KUKA KRL program: MyProgram_251().src

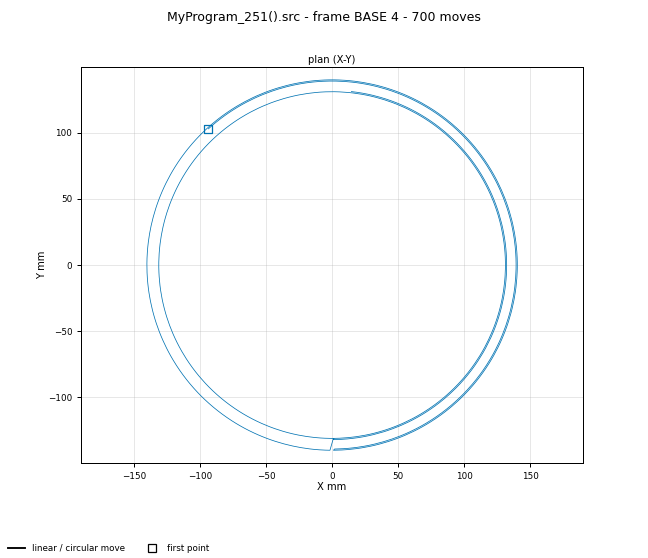
[picture p0: tool path of MyProgram_251().src in frame BASE 4, 700 of 700 moves have a stored position in this frame; points joined in program order, loops and branches not executed]
&ACCESS RVP
&REL 1
&PARAM TEMPLATE = C:\KRC\Roboter\Template\vorgabe
&PARAM EDITMASK = *
DEF MyProgram_251()
; ---- Setting reference (Base) ----
$BASE = BASE_DATA[4]

; --------------------------
; ---- Setting tool (TCP) ----
$TOOL = TOOL_DATA[3]
; --------------------------

$VEL.CP = VEL_APROX_PRINT
Startdeposition()
$VEL.CP = VEL_PRINT
LIN {X -93.5132,Y 103.0033,Z 164,A 132.083,B 11.8455,C 0.0416,E1 11.7391,E2 318.6736} C_DIS
LIN {X -90.9091,Y 105.3089,Z 164,A 130.6284,B 11.8455,C 0.0393,E1 11.7422,E2 320.1295} C_DIS
LIN {X -88.157,Y 107.6233,Z 164,A 129.1078,B 11.8455,C 0.0373,E1 11.7455,E2 321.6535} C_DIS
LIN {X -84.8361,Y 110.2606,Z 164,A 127.2395,B 11.8455,C 0.0369,E1 11.7496,E2 323.535} C_DIS
LIN {X -82.0924,Y 112.3181,Z 164,A 125.9276,B 11.8455,C 0.032,E1 11.7525,E2 324.833} C_DIS
LIN {X -78.8716,Y 114.6024,Z 164,A 124.2342,B 11.8455,C 0.0308,E1 11.7564,E2 326.5331} C_DIS
LIN {X -75.1837,Y 117.055,Z 164,A 121.9812,B 11.8455,C 0.0378,E1 11.7618,E2 328.8371} C_DIS
LIN {X -71.4051,Y 119.3975,Z 164,A 120.7033,B 11.8455,C 0.0219,E1 11.7647,E2 330.0452} C_DIS
LIN {X -67.8999,Y 121.4253,Z 164,A 118.948,B 11.8455,C 0.0214,E1 11.769,E2 331.8098} C_DIS
LIN {X -64.5496,Y 123.2364,Z 164,A 117.0261,B 11.8455,C 0.0276,E1 11.7738,E2 333.7737} C_DIS
LIN {X -61.2678,Y 124.9008,Z 164,A 115.8624,B 11.8455,C 0.0171,E1 11.7766,E2 334.8928} C_DIS
LIN {X -58.3954,Y 126.2689,Z 164,A 114.5881,B 11.8455,C 0.0145,E1 11.7798,E2 336.1615} C_DIS
LIN {X -55.0308,Y 127.7713,Z 164,A 112.9634,B 11.8455,C 0.0152,E1 11.784,E2 337.7981} C_DIS
LIN {X -51.9488,Y 129.055,Z 164,A 111.5636,B 11.8455,C 0.0142,E1 11.7877,E2 339.1998} C_DIS
LIN {X -47.7233,Y 130.6779,Z 164,A 109.8659,B 11.8456,C 0.0081,E1 11.792,E2 340.8755} C_DIS
LIN {X -45.5011,Y 131.4669,Z 164,A 108.7026,B 11.8456,C 0.0118,E1 11.7952,E2 342.0617} C_DIS
LIN {X -40.6187,Y 133.0565,Z 164,A 106.6929,B 11.8456,C 0.0072,E1 11.8005,E2 344.0567} C_DIS
LIN {X -37.3347,Y 134.0151,Z 164,A 105.2264,B 11.8456,C 0.0074,E1 11.8044,E2 345.5294} C_DIS
LIN {X -34.0868,Y 134.8778,Z 164,A 103.8149,B 11.8456,C 0.007,E1 11.8082,E2 346.9433} C_DIS
LIN {X -29.7542,Y 135.8999,Z 164,A 101.958,B 11.8456,C 0.0062,E1 11.8133,E2 348.8019} C_DIS
LIN {X -26.0587,Y 136.6561,Z 164,A 100.4689,B 11.8456,C 0.0037,E1 11.8174,E2 350.2819} C_DIS
LIN {X -22.525,Y 137.2834,Z 164,A 98.5845,B 11.8456,C 0.0129,E1 11.8227,E2 352.2155} C_DIS
LIN {X -18.6482,Y 137.8642,Z 164,A 97.4654,B 11.8456,C -0.0001,E1 11.8256,E2 353.2725} C_DIS
LIN {X -14.4572,Y 138.366,Z 164,A 95.6217,B 11.8456,C 0.0018,E1 11.8308,E2 355.1283} C_DIS
LIN {X -10.8534,Y 138.6965,Z 164,A 94.0872,B 11.8456,C 0.0025,E1 11.835,E2 356.6675} C_DIS
LIN {X -7.1224,Y 138.9363,Z 164,A 92.5483,B 11.8456,C 0.0021,E1 11.8393,E2 358.2053} C_DIS
LIN {X -1.7781,Y 139.1081,Z 164,A 90.2365,B 11.8456,C 0.0046,E1 11.8458,E2 360.5297} C_DIS
LIN {X 2.8679,Y 139.0903,Z 164,A 88.5296,B 11.8456,C -0.0007,E1 11.8505,E2 362.2101} C_DIS
LIN {X 6.3016,Y 138.9776,Z 164,A 87.1185,B 11.8456,C -0.0007,E1 11.8544,E2 363.6202} C_DIS
LIN {X 9.3557,Y 138.8057,Z 164,A 85.6308,B 11.8456,C 0.0053,E1 11.8587,E2 365.1356} C_DIS
LIN {X 15.0229,Y 138.3051,Z 164,A 83.549,B 11.8456,C -0.001,E1 11.8644,E2 367.1842} C_DIS
LIN {X 18.2395,Y 137.9178,Z 164,A 82.134,B 11.8456,C 0.0015,E1 11.8683,E2 368.6087} C_DIS
LIN {X 21.7401,Y 137.4101,Z 164,A 80.0938,B 11.8456,C 0.0172,E1 11.8741,E2 370.7205} C_DIS
LIN {X 26.5047,Y 136.5709,Z 164,A 78.6953,B 11.8456,C 0.0028,E1 11.8778,E2 372.0452} C_DIS
LIN {X 30.1426,Y 135.8161,Z 164,A 77.0002,B 11.8456,C 0.0079,E1 11.8825,E2 373.7605} C_DIS
LIN {X 34.389,Y 134.8012,Z 164,A 75.2809,B 11.8456,C 0.007,E1 11.8871,E2 375.4696} C_DIS
LIN {X 38.2782,Y 133.7512,Z 164,A 73.7125,B 11.8456,C 0.0059,E1 11.8913,E2 377.0265} C_DIS
LIN {X 41.1605,Y 132.8907,Z 164,A 72.462,B 11.8456,C 0.0072,E1 11.8946,E2 378.2782} C_DIS
LIN {X 45.0474,Y 131.6242,Z 164,A 70.7128,B 11.8456,C 0.0104,E1 11.8993,E2 380.0355} C_DIS
LIN {X 48.204,Y 130.5016,Z 164,A 69.5013,B 11.8456,C 0.0072,E1 11.9024,E2 381.2259} C_DIS
LIN {X 50.6781,Y 129.5596,Z 164,A 68.3915,B 11.8456,C 0.0088,E1 11.9053,E2 382.338} C_DIS
LIN {X 53.1807,Y 128.5531,Z 164,A 67.3491,B 11.8456,C 0.0082,E1 11.908,E2 383.3718} C_DIS
LIN {X 57.2624,Y 126.7878,Z 164,A 65.4033,B 11.8456,C 0.0133,E1 11.913,E2 385.3319} C_DIS
LIN {X 60.3441,Y 125.35,Z 164,A 63.9218,B 11.8456,C 0.0172,E1 11.9168,E2 386.8236} C_DIS
LIN {X 64.3775,Y 123.3268,Z 164,A 62.1382,B 11.8456,C 0.0175,E1 11.9212,E2 388.598} C_DIS
LIN {X 68.1253,Y 121.2986,Z 164,A 60.3486,B 11.8456,C 0.0209,E1 11.9256,E2 390.3922} C_DIS
LIN {X 71.8558,Y 119.1267,Z 164,A 58.6255,B 11.8456,C 0.022,E1 11.9297,E2 392.1087} C_DIS
LIN {X 75.3059,Y 116.9767,Z 164,A 56.8769,B 11.8456,C 0.0266,E1 11.9338,E2 393.8669} C_DIS
LIN {X 79.1791,Y 114.3905,Z 164,A 55.0231,B 11.8456,C 0.0279,E1 11.9381,E2 395.7131} C_DIS
LIN {X 82.2792,Y 112.1809,Z 164,A 53.4542,B 11.8456,C 0.0305,E1 11.9416,E2 397.2825} C_DIS
LIN {X 85.5645,Y 109.6965,Z 164,A 51.786,B 11.8456,C 0.0327,E1 11.9453,E2 398.9477} C_DIS
LIN {X 88.6989,Y 107.177,Z 164,A 50.0509,B 11.8456,C 0.0379,E1 11.9491,E2 400.6931} C_DIS
LIN {X 91.429,Y 104.8578,Z 164,A 48.639,B 11.8456,C 0.0389,E1 11.9521,E2 402.0976} C_DIS
LIN {X 94.8874,Y 101.7389,Z 164,A 46.6702,B 11.8456,C 0.0441,E1 11.9561,E2 404.0735} C_DIS
LIN {X 97.912,Y 98.8317,Z 164,A 45.0073,B 11.8456,C 0.0457,E1 11.9595,E2 405.729} C_DIS
LIN {X 101.1689,Y 95.4948,Z 164,A 42.6719,B 11.8454,C 0.0613,E1 11.9641,E2 408.1169} C_DIS
LIN {X 104.3624,Y 91.9942,Z 164,A 41.1925,B 11.8454,C 0.0524,E1 11.9667,E2 409.5385} C_DIS
LIN {X 107.3104,Y 88.5379,Z 164,A 39.3371,B 11.8454,C 0.0561,E1 11.97,E2 411.3929} C_DIS
LIN {X 109.9995,Y 85.1735,Z 164,A 37.6211,B 11.8454,C 0.0585,E1 11.973,E2 413.1027} C_DIS
LIN {X 112.4762,Y 81.8755,Z 164,A 35.9215,B 11.8454,C 0.0625,E1 11.9758,E2 414.8033} C_DIS
LIN {X 114.8679,Y 78.4848,Z 164,A 34.1903,B 11.8454,C 0.0672,E1 11.9786,E2 416.5384} C_DIS
LIN {X 117.2497,Y 74.8796,Z 164,A 32.3977,B 11.8454,C 0.0719,E1 11.9813,E2 418.3338} C_DIS
LIN {X 120.2343,Y 69.9875,Z 164,A 29.8739,B 11.8454,C 0.0824,E1 11.9849,E2 420.8797} C_DIS
LIN {X 121.9796,Y 66.8991,Z 164,A 28.9447,B 11.8454,C 0.071,E1 11.9861,E2 421.7431} C_DIS
LIN {X 123.3941,Y 64.2493,Z 164,A 27.5566,B 11.8454,C 0.0785,E1 11.9879,E2 423.1511} C_DIS
LIN {X 124.8289,Y 61.4135,Z 164,A 26.2825,B 11.8454,C 0.0809,E1 11.9895,E2 424.4218} C_DIS
LIN {X 126.5429,Y 57.8029,Z 164,A 24.4503,B 11.8453,C 0.0906,E1 11.9917,E2 426.2788} C_DIS
LIN {X 129.4436,Y 50.9761,Z 164,A 21.3576,B 11.8452,C 0.0999,E1 11.995,E2 429.3787} C_DIS
LIN {X 131.0516,Y 46.6866,Z 164,A 19.7563,B 11.8452,C 0.0969,E1 11.9965,E2 430.9456} C_DIS
LIN {X 131.9741,Y 44.0084,Z 164,A 18.5216,B 11.8452,C 0.1021,E1 11.9976,E2 432.1899} C_DIS
LIN {X 133.2683,Y 39.9269,Z 164,A 16.8422,B 11.8452,C 0.1046,E1 11.999,E2 433.8604} C_DIS
LIN {X 134.1255,Y 36.94,Z 164,A 15.5694,B 11.8452,C 0.108,E1 12,E2 435.1334} C_DIS
LIN {X 134.9661,Y 33.7389,Z 164,A 14.2687,B 11.8451,C 0.1101,E1 12.0009,E2 436.4275} C_DIS
LIN {X 135.6818,Y 30.7319,Z 164,A 12.9918,B 11.8451,C 0.1138,E1 12.0017,E2 437.706} C_DIS
LIN {X 136.5733,Y 26.4921,Z 164,A 11.3784,B 11.8451,C 0.114,E1 12.0026,E2 439.2995} C_DIS
LIN {X 137.6895,Y 19.8898,Z 164,A 8.3669,B 11.8449,C 0.1294,E1 12.004,E2 442.3459} C_DIS
LIN {X 138.4064,Y 14.0802,Z 164,A 6.13,B 11.8449,C 0.1314,E1 12.0047,E2 444.5633} C_DIS
LIN {X 138.8292,Y 8.9791,Z 164,A 3.8602,B 11.8448,C 0.1423,E1 12.0052,E2 446.8558} C_DIS
LIN {X 139.0245,Y 5.1275,Z 164,A 2.3451,B 11.8448,C 0.1448,E1 12.0053,E2 448.3632} C_DIS
LIN {X 139.1177,Y 0.5934,Z 164,A 0.6055,B 11.8448,C 0.1466,E1 12.0054,E2 450.0885} C_DIS
LIN {X 139.0869,Y -3.0686,Z 164,A -1.0543,B 11.8446,C 0.1555,E1 12.0054,E2 451.7693} C_DIS
LIN {X 138.9554,Y -6.7431,Z 164,A -2.2689,B 11.8446,C 0.1512,E1 12.0052,E2 452.9474} C_DIS
LIN {X 138.8089,Y -9.3088,Z 164,A -3.4315,B 11.8446,C 0.1574,E1 12.005,E2 454.1245} C_DIS
LIN {X 138.443,Y -13.7002,Z 164,A -5.0964,B 11.8446,C 0.1584,E1 12.0046,E2 455.7722} C_DIS
LIN {X 138.1355,Y -16.5095,Z 164,A -6.3924,B 11.8445,C 0.1657,E1 12.0042,E2 457.0864} C_DIS
LIN {X 137.6077,Y -20.4623,Z 164,A -8.0526,B 11.8444,C 0.171,E1 12.0035,E2 458.7507} C_DIS
LIN {X 137.0427,Y -23.9491,Z 164,A -9.9366,B 11.8441,C 0.1878,E1 12.0026,E2 460.6908} C_DIS
LIN {X 136.1753,Y -28.4745,Z 164,A -11.2702,B 11.8443,C 0.1769,E1 12.0019,E2 461.9551} C_DIS
LIN {X 135.5749,Y -31.1998,Z 164,A -12.4598,B 11.8443,C 0.1814,E1 12.0012,E2 463.1511} C_DIS
LIN {X 134.6428,Y -35.0126,Z 164,A -14.1607,B 11.8441,C 0.1886,E1 12,E2 464.8647} C_DIS
LIN {X 133.4452,Y -39.3237,Z 164,A -15.8891,B 11.8441,C 0.1905,E1 11.9987,E2 466.5806} C_DIS
LIN {X 132.2596,Y -43.1508,Z 164,A -17.4741,B 11.8441,C 0.1933,E1 11.9973,E2 468.1593} C_DIS
LIN {X 131.3169,Y -45.9338,Z 164,A -18.779,B 11.8439,C 0.1995,E1 11.9961,E2 469.4777} C_DIS
LIN {X 129.7349,Y -50.2272,Z 164,A -20.3354,B 11.844,C 0.1952,E1 11.9947,E2 470.9943} C_DIS
LIN {X 128.9064,Y -52.3176,Z 164,A -21.5007,B 11.8439,C 0.2048,E1 11.9934,E2 472.1913} C_DIS
LIN {X 127.3612,Y -55.9795,Z 164,A -23.075,B 11.8439,C 0.2075,E1 11.9917,E2 473.7596} C_DIS
LIN {X 125.8906,Y -59.2126,Z 164,A -24.5095,B 11.8438,C 0.2107,E1 11.99,E2 475.1922} C_DIS
LIN {X 123.5041,Y -64.0398,Z 164,A -26.6881,B 11.8437,C 0.2155,E1 11.9873,E2 477.3685} C_DIS
LIN {X 121.613,Y -67.5628,Z 164,A -28.4394,B 11.8435,C 0.2229,E1 11.9849,E2 479.1351} C_DIS
LIN {X 119.3266,Y -71.5241,Z 164,A -30.4512,B 11.8434,C 0.2315,E1 11.982,E2 481.1655} C_DIS
LIN {X 116.6984,Y -75.7357,Z 164,A -32.7824,B 11.8431,C 0.245,E1 11.9785,E2 483.5355} C_DIS
LIN {X 113.9889,Y -79.7564,Z 164,A -34.5272,B 11.8431,C 0.2427,E1 11.9757,E2 485.2506} C_DIS
LIN {X 111.9253,Y -82.6271,Z 164,A -35.7711,B 11.8432,C 0.2402,E1 11.9737,E2 486.4691} C_DIS
LIN {X 108.9221,Y -86.5471,Z 164,A -37.6893,B 11.8432,C 0.2418,E1 11.9704,E2 488.3748} C_DIS
LIN {X 106.4676,Y -89.5493,Z 164,A -39.2737,B 11.8432,C 0.2452,E1 11.9676,E2 489.9594} C_DIS
LIN {X 103.9721,Y -92.4357,Z 164,A -40.8028,B 11.8431,C 0.2476,E1 11.9648,E2 491.4849} C_DIS
LIN {X 102.2519,Y -94.3346,Z 164,A -41.8981,B 11.843,C 0.2511,E1 11.9627,E2 492.5865} C_DIS
LIN {X 99.3369,Y -97.3991,Z 164,A -43.6258,B 11.843,C 0.2546,E1 11.9594,E2 494.3143} C_DIS
LIN {X 96.2847,Y -100.4177,Z 164,A -45.38,B 11.8428,C 0.258,E1 11.9559,E2 496.0687} C_DIS
LIN {X 93.0721,Y -103.4026,Z 164,A -47.1893,B 11.8428,C 0.2619,E1 11.9521,E2 497.8804} C_DIS
LIN {X 89.8236,Y -106.2368,Z 164,A -48.9498,B 11.8427,C 0.265,E1 11.9484,E2 499.6408} C_DIS
LIN {X 86.4839,Y -108.9724,Z 164,A -50.7,B 11.8427,C 0.2677,E1 11.9446,E2 501.3894} C_DIS
LIN {X 82.9756,Y -111.6668,Z 164,A -52.5243,B 11.8425,C 0.2712,E1 11.9405,E2 503.2158} C_DIS
LIN {X 79.1848,Y -114.3866,Z 164,A -54.4412,B 11.8425,C 0.2746,E1 11.9362,E2 505.1341} C_DIS
LIN {X 75.5705,Y -116.8057,Z 164,A -56.1855,B 11.8425,C 0.2764,E1 11.9321,E2 506.8742} C_DIS
LIN {X 71.1252,Y -119.5643,Z 164,A -58.2357,B 11.8425,C 0.277,E1 11.9272,E2 508.913} C_DIS
LIN {X 67.8853,Y -121.4335,Z 164,A -59.88,B 11.8423,C 0.2823,E1 11.9232,E2 510.5722} C_DIS
LIN {X 63.8811,Y -123.5872,Z 164,A -61.6454,B 11.8423,C 0.2821,E1 11.9189,E2 512.3255} C_DIS
LIN {X 58.7901,Y -126.0864,Z 164,A -63.8155,B 11.8423,C 0.2808,E1 11.9135,E2 514.4764} C_DIS
LIN {X 55.0946,Y -127.7438,Z 164,A -65.6415,B 11.8422,C 0.2874,E1 11.9088,E2 516.3242} C_DIS
LIN {X 51.7597,Y -129.1313,Z 164,A -67.194,B 11.8421,C 0.291,E1 11.9047,E2 517.8863} C_DIS
LIN {X 48.2107,Y -130.4991,Z 164,A -68.6428,B 11.8421,C 0.2896,E1 11.901,E2 519.3213} C_DIS
LIN {X 45.2496,Y -131.5541,Z 164,A -70.0506,B 11.8421,C 0.2942,E1 11.8972,E2 520.7447} C_DIS
LIN {X 41.6349,Y -132.744,Z 164,A -71.4992,B 11.8421,C 0.2926,E1 11.8934,E2 522.1794} C_DIS
LIN {X 38.929,Y -133.5607,Z 164,A -72.6474,B 11.8421,C 0.2932,E1 11.8903,E2 523.3264} C_DIS
LIN {X 35.3733,Y -134.547,Z 164,A -74.1782,B 11.842,C 0.2949,E1 11.8862,E2 524.8597} C_DIS
LIN {X 32.2595,Y -135.3269,Z 164,A -75.4773,B 11.842,C 0.2954,E1 11.8827,E2 526.1569} C_DIS
LIN {X 28.5095,Y -136.1682,Z 164,A -77.5593,B 11.8416,C 0.31,E1 11.8768,E2 528.3038} C_DIS
LIN {X 24.3803,Y -136.9656,Z 164,A -78.9498,B 11.8418,C 0.302,E1 11.8731,E2 529.6518} C_DIS
LIN {X 18.9709,Y -137.8208,Z 164,A -81.0414,B 11.8418,C 0.2989,E1 11.8674,E2 531.7239} C_DIS
LIN {X 15.8743,Y -138.2113,Z 164,A -82.7304,B 11.8416,C 0.3103,E1 11.8626,E2 533.4653} C_DIS
LIN {X 12.0921,Y -138.5926,Z 164,A -84.0223,B 11.8418,C 0.3037,E1 11.8591,E2 534.7231} C_DIS
LIN {X 8.5469,Y -138.8559,Z 164,A -85.456,B 11.8418,C 0.3033,E1 11.8551,E2 536.1537} C_DIS
LIN {X 4.8994,Y -139.0334,Z 164,A -86.8146,B 11.8418,C 0.2999,E1 11.8513,E2 537.4945} C_DIS
LIN {X 1.8653,Y -139.107,Z 164,A -88.1849,B 11.8418,C 0.3033,E1 11.8475,E2 538.8809} C_DIS
LIN {X 1.8653,Y -139.107,Z 164,A -88.1849,B 11.8418,C 0.3033,E1 11.8475,E2 538.8809} C_DIS
Enddeposition()
LIN {X 1.0011,Y -140.0329,Z 164,A -87.9487,B 11.842,C 0.2948,E1 11.8483,E2 538.6034} C_DIS
Startdeposition()
$VEL.CP = VEL_PRINT
LIN {X 4.0661,Y -139.9794,Z 164,A -86.5813,B 11.8421,C 0.2915,E1 11.8522,E2 537.2207} C_DIS
LIN {X 7.3718,Y -139.8446,Z 164,A -85.0824,B 11.8422,C 0.2872,E1 11.8564,E2 535.702} C_DIS
LIN {X 12.0541,Y -139.5188,Z 164,A -83.2838,B 11.8422,C 0.2898,E1 11.8614,E2 533.9183} C_DIS
LIN {X 15.6406,Y -139.1636,Z 164,A -81.8412,B 11.8422,C 0.29,E1 11.8654,E2 532.4791} C_DIS
LIN {X 18.9541,Y -138.7517,Z 164,A -80.3719,B 11.8422,C 0.2865,E1 11.8695,E2 530.9954} C_DIS
LIN {X 22.2682,Y -138.2586,Z 164,A -79.0797,B 11.8422,C 0.2879,E1 11.873,E2 529.7126} C_DIS
LIN {X 25.6653,Y -137.6676,Z 164,A -77.6805,B 11.8422,C 0.2873,E1 11.8768,E2 528.314} C_DIS
LIN {X 29.0223,Y -136.9988,Z 164,A -76.2843,B 11.8422,C 0.2863,E1 11.8807,E2 526.9174} C_DIS
LIN {X 32.3823,Y -136.2433,Z 164,A -74.8831,B 11.8422,C 0.2854,E1 11.8845,E2 525.5162} C_DIS
LIN {X 35.7212,Y -135.406,Z 164,A -73.4347,B 11.8423,C 0.2831,E1 11.8884,E2 524.0615} C_DIS
LIN {X 39.0397,Y -134.4866,Z 164,A -72.0852,B 11.8423,C 0.2834,E1 11.892,E2 522.7187} C_DIS
LIN {X 42.3077,Y -133.4945,Z 164,A -70.6887,B 11.8423,C 0.282,E1 11.8957,E2 521.3212} C_DIS
LIN {X 45.5732,Y -132.4152,Z 164,A -69.2884,B 11.8423,C 0.2807,E1 11.8995,E2 519.9207} C_DIS
LIN {X 48.8112,Y -131.2562,Z 164,A -67.8889,B 11.8424,C 0.2793,E1 11.9031,E2 518.5211} C_DIS
LIN {X 52.0199,Y -130.0179,Z 164,A -66.4897,B 11.8424,C 0.2779,E1 11.9068,E2 517.1217} C_DIS
LIN {X 55.1975,Y -128.7012,Z 164,A -65.0964,B 11.8424,C 0.2765,E1 11.9103,E2 515.729} C_DIS
LIN {X 58.3787,Y -127.2899,Z 164,A -63.6912,B 11.8425,C 0.2751,E1 11.9139,E2 514.3251} C_DIS
LIN {X 61.4407,Y -125.841,Z 164,A -62.301,B 11.8425,C 0.273,E1 11.9174,E2 512.933} C_DIS
LIN {X 64.5115,Y -124.2952,Z 164,A -60.9185,B 11.8425,C 0.2717,E1 11.9209,E2 511.5524} C_DIS
LIN {X 67.544,Y -122.6746,Z 164,A -59.4693,B 11.8427,C 0.2683,E1 11.9244,E2 510.0963} C_DIS
LIN {X 71.2578,Y -120.5554,Z 164,A -57.7572,B 11.8427,C 0.2666,E1 11.9286,E2 508.3875} C_DIS
LIN {X 74.4296,Y -118.6234,Z 164,A -56.1383,B 11.8428,C 0.2612,E1 11.9324,E2 506.7541} C_DIS
LIN {X 78.2094,Y -116.166,Z 164,A -54.3438,B 11.8428,C 0.2594,E1 11.9366,E2 504.9642} C_DIS
LIN {X 81.8544,Y -113.6273,Z 164,A -52.5667,B 11.8429,C 0.2573,E1 11.9406,E2 503.1906} C_DIS
LIN {X 84.813,Y -111.4361,Z 164,A -51.1314,B 11.8429,C 0.2565,E1 11.9438,E2 501.7631} C_DIS
LIN {X 87.5061,Y -109.3341,Z 164,A -49.6095,B 11.8431,C 0.2502,E1 11.9472,E2 500.2235} C_DIS
LIN {X 91.0025,Y -106.4417,Z 164,A -47.7743,B 11.8431,C 0.2471,E1 11.9511,E2 498.3891} C_DIS
LIN {X 94.4857,Y -103.3621,Z 164,A -45.953,B 11.8431,C 0.2455,E1 11.9549,E2 496.5763} C_DIS
LIN {X 97.1954,Y -100.818,Z 164,A -44.378,B 11.8432,C 0.2407,E1 11.9581,E2 494.9925} C_DIS
LIN {X 100.2454,Y -97.7862,Z 164,A -42.7214,B 11.8432,C 0.2399,E1 11.9613,E2 493.3475} C_DIS
LIN {X 103.184,Y -94.6795,Z 164,A -40.9463,B 11.8434,C 0.2352,E1 11.9647,E2 491.5671} C_DIS
LIN {X 106.0445,Y -91.4643,Z 164,A -39.1946,B 11.8434,C 0.2314,E1 11.9679,E2 489.8145} C_DIS
LIN {X 108.8027,Y -88.1658,Z 164,A -37.5509,B 11.8434,C 0.2306,E1 11.9708,E2 488.184} C_DIS
LIN {X 111.2882,Y -85.0063,Z 164,A -35.8382,B 11.8436,C 0.2247,E1 11.9738,E2 486.4605} C_DIS
LIN {X 114.0144,Y -81.3135,Z 164,A -33.9826,B 11.8436,C 0.2207,E1 11.9768,E2 484.6057} C_DIS
LIN {X 116.4423,Y -77.7967,Z 164,A -32.2283,B 11.8437,C 0.2161,E1 11.9796,E2 482.8485} C_DIS
LIN {X 118.7733,Y -74.1897,Z 164,A -30.5934,B 11.8437,C 0.2152,E1 11.982,E2 481.2276} C_DIS
LIN {X 120.5616,Y -71.2473,Z 164,A -29.2021,B 11.8437,C 0.2121,E1 11.984,E2 479.837} C_DIS
LIN {X 122.2757,Y -68.2639,Z 164,A -27.8008,B 11.8438,C 0.2086,E1 11.9859,E2 478.4348} C_DIS
LIN {X 124.0773,Y -64.9264,Z 164,A -26.3319,B 11.8438,C 0.2069,E1 11.9878,E2 476.9749} C_DIS
LIN {X 125.483,Y -62.1664,Z 164,A -25.0269,B 11.844,C 0.2023,E1 11.9895,E2 475.6634} C_DIS
LIN {X 126.9611,Y -59.0896,Z 164,A -23.6411,B 11.844,C 0.1989,E1 11.9911,E2 474.2774} C_DIS
LIN {X 128.3961,Y -55.9032,Z 164,A -22.2202,B 11.844,C 0.1952,E1 11.9927,E2 472.856} C_DIS
LIN {X 129.7483,Y -52.6888,Z 164,A -20.8116,B 11.8441,C 0.1918,E1 11.9942,E2 471.448} C_DIS
LIN {X 131.0142,Y -49.4571,Z 164,A -19.4104,B 11.8441,C 0.1884,E1 11.9956,E2 470.0476} C_DIS
LIN {X 132.1942,Y -46.2107,Z 164,A -18.0021,B 11.8442,C 0.1845,E1 11.997,E2 468.6384} C_DIS
LIN {X 133.29,Y -42.9479,Z 164,A -16.6248,B 11.8442,C 0.1814,E1 11.9982,E2 467.2634} C_DIS
LIN {X 134.3017,Y -39.671,Z 164,A -15.2396,B 11.8443,C 0.1779,E1 11.9993,E2 465.8789} C_DIS
LIN {X 135.2298,Y -36.3818,Z 164,A -13.8591,B 11.8443,C 0.1744,E1 12.0003,E2 464.499} C_DIS
LIN {X 136.0738,Y -33.0855,Z 164,A -12.4855,B 11.8444,C 0.171,E1 12.0012,E2 463.1263} C_DIS
LIN {X 136.8606,Y -29.6623,Z 164,A -11.0984,B 11.8444,C 0.1683,E1 12.0021,E2 461.744} C_DIS
LIN {X 137.5057,Y -26.5124,Z 164,A -9.7798,B 11.8445,C 0.1643,E1 12.0028,E2 460.4235} C_DIS
LIN {X 138.0567,Y -23.4777,Z 164,A -8.6616,B 11.8445,C 0.1649,E1 12.0033,E2 459.3225} C_DIS
LIN {X 138.5281,Y -20.5222,Z 164,A -7.2952,B 11.8446,C 0.1571,E1 12.0039,E2 457.9363} C_DIS
LIN {X 139.0402,Y -16.6892,Z 164,A -5.7109,B 11.8446,C 0.1524,E1 12.0045,E2 456.3499} C_DIS
LIN {X 139.4224,Y -13.1212,Z 164,A -4.3109,B 11.8447,C 0.1501,E1 12.0049,E2 454.9572} C_DIS
LIN {X 139.6938,Y -9.8232,Z 164,A -2.8259,B 11.8448,C 0.1422,E1 12.0052,E2 453.4536} C_DIS
LIN {X 139.9446,Y -5.1342,Z 164,A -1.0609,B 11.8448,C 0.1411,E1 12.0054,E2 451.7067} C_DIS
LIN {X 140.0311,Y -1.6039,Z 164,A 0.4767,B 11.8449,C 0.1341,E1 12.0054,E2 450.1556} C_DIS
LIN {X 140.0178,Y 2.3995,Z 164,A 1.9711,B 11.8449,C 0.1335,E1 12.0054,E2 448.678} C_DIS
LIN {X 139.9217,Y 5.7199,Z 164,A 3.3076,B 11.8449,C 0.1302,E1 12.0053,E2 447.343} C_DIS
LIN {X 139.6938,Y 9.8232,Z 164,A 4.9783,B 11.845,C 0.1256,E1 12.005,E2 445.672} C_DIS
LIN {X 139.3653,Y 13.7165,Z 164,A 6.5723,B 11.845,C 0.121,E1 12.0046,E2 444.0769} C_DIS
LIN {X 138.9675,Y 17.2987,Z 164,A 8.0038,B 11.845,C 0.118,E1 12.0041,E2 442.6496} C_DIS
LIN {X 138.4725,Y 20.8891,Z 164,A 9.3879,B 11.845,C 0.1166,E1 12.0036,E2 441.2766} C_DIS
LIN {X 137.9729,Y 23.9718,Z 164,A 10.7556,B 11.8452,C 0.1102,E1 12.0029,E2 439.8961} C_DIS
LIN {X 137.3429,Y 27.3482,Z 164,A 12.1426,B 11.8452,C 0.1067,E1 12.0022,E2 438.5101} C_DIS
LIN {X 136.6336,Y 30.6945,Z 164,A 13.5971,B 11.8452,C 0.101,E1 12.0013,E2 437.0471} C_DIS
LIN {X 135.8381,Y 34.0415,Z 164,A 14.9103,B 11.8452,C 0.0998,E1 12.0005,E2 435.7448} C_DIS
LIN {X 134.8789,Y 37.6608,Z 164,A 16.3541,B 11.8452,C 0.0981,E1 11.9994,E2 434.311} C_DIS
LIN {X 134.0008,Y 40.6759,Z 164,A 17.6916,B 11.8453,C 0.0929,E1 11.9983,E2 432.9656} C_DIS
LIN {X 132.9613,Y 43.9545,Z 164,A 19.0814,B 11.8453,C 0.0895,E1 11.9972,E2 431.5767} C_DIS
LIN {X 131.8417,Y 47.2066,Z 164,A 20.4792,B 11.8453,C 0.0859,E1 11.9959,E2 430.1789} C_DIS
LIN {X 130.6397,Y 50.4379,Z 164,A 21.8643,B 11.8453,C 0.0828,E1 11.9945,E2 428.796} C_DIS
LIN {X 129.3643,Y 53.6248,Z 164,A 23.2505,B 11.8453,C 0.0795,E1 11.993,E2 427.4109} C_DIS
LIN {X 128.0141,Y 56.7731,Z 164,A 24.6345,B 11.8454,C 0.0763,E1 11.9915,E2 426.0281} C_DIS
LIN {X 126.5828,Y 59.8969,Z 164,A 26.0177,B 11.8454,C 0.0732,E1 11.9899,E2 424.6467} C_DIS
LIN {X 125.0848,Y 62.9664,Z 164,A 27.4051,B 11.8454,C 0.0699,E1 11.9881,E2 423.2595} C_DIS
LIN {X 123.5011,Y 66.0205,Z 164,A 28.8037,B 11.8454,C 0.0665,E1 11.9863,E2 421.8611} C_DIS
LIN {X 121.8363,Y 69.0451,Z 164,A 30.1977,B 11.8454,C 0.0635,E1 11.9844,E2 420.4685} C_DIS
LIN {X 120.1015,Y 72.0202,Z 164,A 31.6257,B 11.8455,C 0.0594,E1 11.9824,E2 419.0371} C_DIS
LIN {X 117.8374,Y 75.6672,Z 164,A 33.4042,B 11.8455,C 0.0544,E1 11.9797,E2 417.2546} C_DIS
LIN {X 115.4743,Y 79.2264,Z 164,A 35.1614,B 11.8455,C 0.05,E1 11.977,E2 415.495} C_DIS
LIN {X 112.9875,Y 82.7346,Z 164,A 36.8825,B 11.8455,C 0.0469,E1 11.9742,E2 413.7778} C_DIS
LIN {X 110.3941,Y 86.1653,Z 164,A 38.5503,B 11.8455,C 0.0455,E1 11.9713,E2 412.1209} C_DIS
LIN {X 108.1182,Y 89.0043,Z 164,A 40.1507,B 11.8455,C 0.039,E1 11.9685,E2 410.5053} C_DIS
LIN {X 105.1528,Y 92.4886,Z 164,A 41.957,B 11.8456,C 0.0368,E1 11.9652,E2 408.7065} C_DIS
LIN {X 102.1494,Y 95.7956,Z 164,A 43.7304,B 11.8456,C 0.0344,E1 11.9619,E2 406.9392} C_DIS
LIN {X 99.6254,Y 98.4179,Z 164,A 45.1621,B 11.8456,C 0.033,E1 11.9591,E2 405.5141} C_DIS
LIN {X 97.1779,Y 100.8349,Z 164,A 46.6112,B 11.8456,C 0.029,E1 11.9562,E2 404.0591} C_DIS
LIN {X 94.0343,Y 103.7723,Z 164,A 48.3899,B 11.8456,C 0.025,E1 11.9525,E2 402.2775} C_DIS
LIN {X 90.8018,Y 106.6123,Z 164,A 50.1534,B 11.8456,C 0.0216,E1 11.9488,E2 400.5129} C_DIS
LIN {X 87.5052,Y 109.3349,Z 164,A 51.781,B 11.8456,C 0.0219,E1 11.9453,E2 398.9004} C_DIS
LIN {X 84.2284,Y 111.8782,Z 164,A 53.5432,B 11.8456,C 0.0171,E1 11.9414,E2 397.1293} C_DIS
LIN {X 80.6289,Y 114.4994,Z 164,A 55.3622,B 11.8456,C 0.0142,E1 11.9372,E2 395.3103} C_DIS
LIN {X 77.074,Y 116.922,Z 164,A 57.1302,B 11.8456,C 0.0111,E1 11.9331,E2 393.5409} C_DIS
LIN {X 73.4459,Y 119.2347,Z 164,A 58.7726,B 11.8456,C 0.0118,E1 11.9293,E2 391.9132} C_DIS
LIN {X 70.4949,Y 121.0031,Z 164,A 60.1681,B 11.8456,C 0.0101,E1 11.9259,E2 390.5191} C_DIS
LIN {X 67.5221,Y 122.6867,Z 164,A 61.5688,B 11.8456,C 0.008,E1 11.9225,E2 389.1178} C_DIS
LIN {X 64.4876,Y 124.3077,Z 164,A 62.9964,B 11.8456,C 0.0056,E1 11.919,E2 387.6875} C_DIS
LIN {X 61.1115,Y 126.0026,Z 164,A 64.6366,B 11.8456,C 0.0011,E1 11.9148,E2 386.0352} C_DIS
LIN {X 57.5135,Y 127.6829,Z 164,A 66.1261,B 11.8456,C 0.0029,E1 11.9111,E2 384.5628} C_DIS
LIN {X 54.2997,Y 129.0824,Z 164,A 67.5486,B 11.8456,C 0.0016,E1 11.9074,E2 383.1418} C_DIS
LIN {X 51.0779,Y 130.3909,Z 164,A 68.9641,B 11.8456,C 0.0004,E1 11.9038,E2 381.7273} C_DIS
LIN {X 47.8376,Y 131.6142,Z 164,A 70.3745,B 11.8456,C -0.0008,E1 11.9001,E2 380.3178} C_DIS
LIN {X 44.5798,Y 132.7531,Z 164,A 71.7801,B 11.8456,C -0.0019,E1 11.8964,E2 378.9131} C_DIS
LIN {X 41.3072,Y 133.8075,Z 164,A 73.2378,B 11.8456,C -0.0045,E1 11.8925,E2 377.4491} C_DIS
LIN {X 37.3328,Y 134.9706,Z 164,A 74.8872,B 11.8456,C -0.0045,E1 11.8881,E2 375.8057} C_DIS
LIN {X 33.7943,Y 135.9009,Z 164,A 76.3563,B 11.8456,C -0.0048,E1 11.8841,E2 374.3404} C_DIS
LIN {X 30.4913,Y 136.6801,Z 164,A 77.8112,B 11.8456,C -0.0074,E1 11.8801,E2 372.8774} C_DIS
LIN {X 26.5137,Y 137.5054,Z 164,A 79.3913,B 11.8456,C -0.0061,E1 11.8758,E2 371.3081} C_DIS
LIN {X 23.4452,Y 138.0622,Z 164,A 80.5265,B 11.8456,C -0.0029,E1 11.8727,E2 370.191} C_DIS
LIN {X 20.5335,Y 138.5265,Z 164,A 81.8972,B 11.8456,C -0.0077,E1 11.8689,E2 368.7999} C_DIS
LIN {X 17.1045,Y 138.9907,Z 164,A 83.3673,B 11.8456,C -0.0096,E1 11.8648,E2 367.3234} C_DIS
LIN {X 13.1184,Y 139.4227,Z 164,A 84.9212,B 11.8456,C -0.0078,E1 11.8605,E2 365.781} C_DIS
LIN {X 9.8203,Y 139.694,Z 164,A 86.4239,B 11.8456,C -0.0119,E1 11.8563,E2 364.2601} C_DIS
LIN {X 5.1216,Y 139.945,Z 164,A 88.2135,B 11.8456,C -0.0085,E1 11.8513,E2 362.4884} C_DIS
LIN {X 1.6056,Y 140.031,Z 164,A 89.7805,B 11.8456,C -0.0118,E1 11.8469,E2 360.9059} C_DIS
LIN {X -2.3939,Y 140.0179,Z 164,A 91.2798,B 11.8456,C -0.0081,E1 11.8428,E2 359.4246} C_DIS
LIN {X -5.7206,Y 139.9217,Z 164,A 92.6362,B 11.8456,C -0.0077,E1 11.839,E2 358.0696} C_DIS
LIN {X -9.8203,Y 139.694,Z 164,A 94.4421,B 11.8456,C -0.0106,E1 11.8339,E2 356.2487} C_DIS
LIN {X -13.9852,Y 139.3395,Z 164,A 96.0303,B 11.8456,C -0.0069,E1 11.8296,E2 354.6768} C_DIS
LIN {X -17.3002,Y 138.9673,Z 164,A 97.5131,B 11.8456,C -0.0093,E1 11.8254,E2 353.18} C_DIS
LIN {X -20.9656,Y 138.4606,Z 164,A 98.7994,B 11.8456,C -0.0028,E1 11.8219,E2 351.9233} C_DIS
LIN {X -23.9569,Y 137.9756,Z 164,A 100.1858,B 11.8456,C -0.0058,E1 11.8181,E2 350.5193} C_DIS
LIN {X -27.3416,Y 137.3443,Z 164,A 101.5945,B 11.8456,C -0.005,E1 11.8142,E2 349.1115} C_DIS
LIN {X -30.7073,Y 136.6307,Z 164,A 103.0041,B 11.8456,C -0.0041,E1 11.8104,E2 347.7026} C_DIS
LIN {X -34.0541,Y 135.8349,Z 164,A 104.4143,B 11.8456,C -0.0031,E1 11.8065,E2 346.293} C_DIS
LIN {X -37.3832,Y 134.9565,Z 164,A 105.8272,B 11.8456,C -0.002,E1 11.8027,E2 344.8806} C_DIS
LIN {X -40.6693,Y 134.0028,Z 164,A 107.2318,B 11.8456,C -0.0009,E1 11.799,E2 343.4765} C_DIS
LIN {X -43.9472,Y 132.9638,Z 164,A 108.6438,B 11.8456,C 0.0004,E1 11.7952,E2 342.0649} C_DIS
LIN {X -47.198,Y 131.8448,Z 164,A 110.056,B 11.8456,C 0.0017,E1 11.7915,E2 340.6531} C_DIS
LIN {X -50.4202,Y 130.6465,Z 164,A 111.4686,B 11.8456,C 0.0031,E1 11.7878,E2 339.241} C_DIS
LIN {X -53.6124,Y 129.3695,Z 164,A 112.8835,B 11.8456,C 0.0045,E1 11.7842,E2 337.8262} C_DIS
LIN {X -56.7574,Y 128.0211,Z 164,A 114.2881,B 11.8456,C 0.0062,E1 11.7806,E2 336.4222} C_DIS
LIN {X -59.8848,Y 126.5886,Z 164,A 115.715,B 11.8456,C 0.0075,E1 11.7769,E2 334.9941} C_DIS
LIN {X -63.0165,Y 125.0593,Z 164,A 117.1353,B 11.8456,C 0.0096,E1 11.7734,E2 333.5758} C_DIS
LIN {X -66.0519,Y 123.4843,Z 164,A 118.5452,B 11.8456,C 0.0113,E1 11.7699,E2 332.1658} C_DIS
LIN {X -69.0578,Y 121.829,Z 164,A 119.9535,B 11.8456,C 0.0133,E1 11.7665,E2 330.7583} C_DIS
LIN {X -71.9999,Y 120.1136,Z 164,A 121.3996,B 11.8456,C 0.0142,E1 11.763,E2 329.3068} C_DIS
LIN {X -75.6548,Y 117.8453,Z 164,A 123.2113,B 11.8456,C 0.0158,E1 11.7587,E2 327.4903} C_DIS
LIN {X -79.237,Y 115.4671,Z 164,A 125.0062,B 11.8456,C 0.018,E1 11.7546,E2 325.6926} C_DIS
LIN {X -82.744,Y 112.9805,Z 164,A 126.6789,B 11.8456,C 0.0232,E1 11.7508,E2 324.0326} C_DIS
LIN {X -85.4965,Y 110.9127,Z 164,A 128.0961,B 11.8456,C 0.0256,E1 11.7476,E2 322.6157} C_DIS
LIN {X -88.1767,Y 108.7939,Z 164,A 129.561,B 11.8456,C 0.0266,E1 11.7444,E2 321.1439} C_DIS
LIN {X -91.4755,Y 106.0348,Z 164,A 131.3717,B 11.8456,C 0.0288,E1 11.7406,E2 319.3285} C_DIS
LIN {X -94.6912,Y 103.1733,Z 164,A 133.161,B 11.8456,C 0.0317,E1 11.7369,E2 317.5375} C_DIS
LIN {X -97.8136,Y 100.2185,Z 164,A 134.8304,B 11.8456,C 0.0376,E1 11.7335,E2 315.8814} C_DIS
LIN {X -100.2458,Y 97.7858,Z 164,A 136.3006,B 11.8456,C 0.0391,E1 11.7306,E2 314.4048} C_DIS
LIN {X -103.184,Y 94.6795,Z 164,A 138.1102,B 11.8456,C 0.0415,E1 11.7272,E2 312.5895} C_DIS
LIN {X -106.0503,Y 91.4575,Z 164,A 139.8988,B 11.8456,C 0.045,E1 11.7239,E2 310.7998} C_DIS
LIN {X -108.8052,Y 88.1627,Z 164,A 141.5748,B 11.8456,C 0.051,E1 11.7209,E2 309.1361} C_DIS
LIN {X -111.2732,Y 85.026,Z 164,A 143.3166,B 11.8456,C 0.0523,E1 11.7179,E2 307.3823} C_DIS
LIN {X -114.0099,Y 81.3197,Z 164,A 145.2157,B 11.8456,C 0.0565,E1 11.7148,E2 305.4836} C_DIS
LIN {X -116.4397,Y 77.8006,Z 164,A 147.0094,B 11.8456,C 0.0598,E1 11.712,E2 303.6863} C_DIS
LIN {X -118.7751,Y 74.1868,Z 164,A 148.6819,B 11.8455,C 0.0663,E1 11.7095,E2 302.027} C_DIS
LIN {X -120.5617,Y 71.247,Z 164,A 150.1039,B 11.8455,C 0.0696,E1 11.7075,E2 300.6048} C_DIS
LIN {X -122.2757,Y 68.2638,Z 164,A 151.5373,B 11.8455,C 0.0727,E1 11.7055,E2 299.1698} C_DIS
LIN {X -124.1052,Y 64.8733,Z 164,A 153.0549,B 11.8455,C 0.0782,E1 11.7035,E2 297.6613} C_DIS
LIN {X -125.4784,Y 62.1757,Z 164,A 154.3714,B 11.8454,C 0.0797,E1 11.7019,E2 296.3365} C_DIS
LIN {X -126.9574,Y 59.0976,Z 164,A 155.791,B 11.8454,C 0.083,E1 11.7002,E2 294.9157} C_DIS
LIN {X -128.3961,Y 55.9032,Z 164,A 157.2491,B 11.8454,C 0.0863,E1 11.6985,E2 293.4561} C_DIS
LIN {X -129.7483,Y 52.6888,Z 164,A 158.692,B 11.8454,C 0.0899,E1 11.697,E2 292.0129} C_DIS
LIN {X -131.0142,Y 49.4571,Z 164,A 160.1273,B 11.8453,C 0.0935,E1 11.6955,E2 290.5773} C_DIS
LIN {X -132.1942,Y 46.2107,Z 164,A 161.557,B 11.8453,C 0.0971,E1 11.6942,E2 289.1471} C_DIS
LIN {X -133.29,Y 42.9479,Z 164,A 163.0137,B 11.8453,C 0.0999,E1 11.6929,E2 287.6859} C_DIS
LIN {X -134.3017,Y 39.671,Z 164,A 164.4015,B 11.8453,C 0.1043,E1 11.6918,E2 286.3018} C_DIS
LIN {X -135.2298,Y 36.3818,Z 164,A 165.8169,B 11.8452,C 0.1079,E1 11.6908,E2 284.8858} C_DIS
LIN {X -136.0738,Y 33.0855,Z 164,A 167.225,B 11.8452,C 0.1115,E1 11.6898,E2 283.4773} C_DIS
LIN {X -136.8327,Y 29.7916,Z 164,A 168.6223,B 11.8452,C 0.1152,E1 11.689,E2 282.0797} C_DIS
LIN {X -137.5057,Y 26.5124,Z 164,A 169.9995,B 11.8451,C 0.119,E1 11.6882,E2 280.7032} C_DIS
LIN {X -138.0567,Y 23.4777,Z 164,A 171.1455,B 11.8451,C 0.1254,E1 11.6877,E2 279.5734} C_DIS
LIN {X -138.5278,Y 20.5244,Z 164,A 172.5468,B 11.8451,C 0.1249,E1 11.6871,E2 278.1509} C_DIS
LIN {X -138.9896,Y 17.1133,Z 164,A 173.98,B 11.845,C 0.1285,E1 11.6865,E2 276.7161} C_DIS
LIN {X -139.3717,Y 13.6499,Z 164,A 175.4877,B 11.845,C 0.1308,E1 11.6861,E2 275.1995} C_DIS
LIN {X -139.6938,Y 9.8232,Z 164,A 177.1328,B 11.845,C 0.1337,E1 11.6858,E2 273.5468} C_DIS
LIN {X -139.9456,Y 5.108,Z 164,A 179.0237,B 11.8448,C 0.1404,E1 11.6855,E2 271.6633} C_DIS
LIN {X -140.0352,Y 0.9249,Z 164,A -179.2844,B 11.8448,C 0.1459,E1 11.6855,E2 269.9758} C_DIS
LIN {X -140.0178,Y -2.3995,Z 164,A -177.9467,B 11.8448,C 0.1504,E1 11.6855,E2 268.6424} C_DIS
LIN {X -139.9217,Y -5.7199,Z 164,A -176.5756,B 11.8447,C 0.1541,E1 11.6856,E2 267.2711} C_DIS
LIN {X -139.6938,Y -9.8232,Z 164,A -174.8622,B 11.8447,C 0.1583,E1 11.6859,E2 265.5555} C_DIS
LIN {X -139.3651,Y -13.7185,Z 164,A -173.2266,B 11.8446,C 0.1622,E1 11.6864,E2 263.9169} C_DIS
LIN {X -138.9675,Y -17.2987,Z 164,A -171.7591,B 11.8446,C 0.1667,E1 11.6868,E2 262.4518} C_DIS
LIN {X -138.4725,Y -20.8891,Z 164,A -170.3411,B 11.8444,C 0.1725,E1 11.6874,E2 261.0435} C_DIS
LIN {X -137.911,Y -24.3181,Z 164,A -168.7679,B 11.8444,C 0.1731,E1 11.6881,E2 259.4523} C_DIS
LIN {X -137.3421,Y -27.3525,Z 164,A -167.515,B 11.8444,C 0.1769,E1 11.6888,E2 258.2019} C_DIS
LIN {X -136.5448,Y -31.0836,Z 164,A -166.0421,B 11.8443,C 0.1834,E1 11.6897,E2 256.7418} C_DIS
LIN {X -135.8383,Y -34.0407,Z 164,A -164.6768,B 11.8443,C 0.1842,E1 11.6906,E2 255.3621} C_DIS
LIN {X -134.959,Y -37.3744,Z 164,A -163.252,B 11.8442,C 0.1878,E1 11.6916,E2 253.9368} C_DIS
LIN {X -134.0006,Y -40.6766,Z 164,A -161.8288,B 11.8442,C 0.1914,E1 11.6928,E2 252.5128} C_DIS
LIN {X -132.9616,Y -43.9537,Z 164,A -160.4058,B 11.8441,C 0.1949,E1 11.694,E2 251.089} C_DIS
LIN {X -131.8425,Y -47.2044,Z 164,A -158.983,B 11.8441,C 0.1984,E1 11.6953,E2 249.6652} C_DIS
LIN {X -130.6528,Y -50.4042,Z 164,A -157.5686,B 11.844,C 0.2018,E1 11.6967,E2 248.2498} C_DIS
LIN {X -129.3729,Y -53.6042,Z 164,A -156.0809,B 11.844,C 0.2037,E1 11.6983,E2 246.7532} C_DIS
LIN {X -128.0153,Y -56.7703,Z 164,A -154.7198,B 11.8438,C 0.2086,E1 11.6998,E2 245.3995} C_DIS
LIN {X -126.5828,Y -59.8969,Z 164,A -153.3056,B 11.8438,C 0.2122,E1 11.7015,E2 243.9855} C_DIS
LIN {X -125.085,Y -62.966,Z 164,A -151.8868,B 11.8438,C 0.2153,E1 11.7032,E2 242.5651} C_DIS
LIN {X -123.5013,Y -66.0201,Z 164,A -150.4605,B 11.8437,C 0.2184,E1 11.7051,E2 241.1374} C_DIS
LIN {X -121.8423,Y -69.0346,Z 164,A -149.0346,B 11.8437,C 0.2216,E1 11.707,E2 239.7101} C_DIS
LIN {X -120.1089,Y -72.0078,Z 164,A -147.4776,B 11.8437,C 0.2216,E1 11.7093,E2 238.1349} C_DIS
LIN {X -117.6449,Y -75.9667,Z 164,A -145.581,B 11.8435,C 0.2264,E1 11.7121,E2 236.241} C_DIS
LIN {X -115.1598,Y -79.6836,Z 164,A -143.7674,B 11.8435,C 0.2311,E1 11.715,E2 234.4307} C_DIS
LIN {X -112.6245,Y -83.2286,Z 164,A -141.9116,B 11.8434,C 0.2335,E1 11.718,E2 232.5665} C_DIS
LIN {X -109.8625,Y -86.8422,Z 164,A -140.1457,B 11.8433,C 0.24,E1 11.721,E2 230.8139} C_DIS
LIN {X -107.5251,Y -89.7197,Z 164,A -138.5002,B 11.8433,C 0.2402,E1 11.724,E2 229.1526} C_DIS
LIN {X -104.5575,Y -93.1611,Z 164,A -136.6676,B 11.8432,C 0.2449,E1 11.7273,E2 227.3244} C_DIS
LIN {X -101.5402,Y -96.4413,Z 164,A -134.8676,B 11.8431,C 0.2492,E1 11.7308,E2 225.5283} C_DIS
LIN {X -99.019,Y -99.0281,Z 164,A -133.4072,B 11.8431,C 0.2526,E1 11.7336,E2 224.0708} C_DIS
LIN {X -96.3989,Y -101.5803,Z 164,A -131.7758,B 11.8431,C 0.2522,E1 11.7369,E2 222.4225} C_DIS
LIN {X -93.0233,Y -104.6801,Z 164,A -129.9369,B 11.8429,C 0.2567,E1 11.7407,E2 220.589} C_DIS
LIN {X -89.7232,Y -107.5222,Z 164,A -128.1577,B 11.8429,C 0.26,E1 11.7445,E2 218.8108} C_DIS
LIN {X -86.482,Y -110.1454,Z 164,A -126.4341,B 11.8428,C 0.2625,E1 11.7483,E2 217.0854} C_DIS
LIN {X -83.2288,Y -112.6244,Z 164,A -124.6888,B 11.8428,C 0.2635,E1 11.7522,E2 215.3311} C_DIS
LIN {X -79.5308,Y -115.2654,Z 164,A -122.8606,B 11.8427,C 0.2672,E1 11.7564,E2 213.5075} C_DIS
LIN {X -75.8378,Y -117.7282,Z 164,A -121.0582,B 11.8427,C 0.2703,E1 11.7606,E2 211.7072} C_DIS
LIN {X -72.7125,Y -119.6834,Z 164,A -119.5998,B 11.8425,C 0.2738,E1 11.7641,E2 210.2555} C_DIS
LIN {X -69.7717,Y -121.4217,Z 164,A -118.1802,B 11.8425,C 0.2751,E1 11.7675,E2 208.8332} C_DIS
LIN {X -66.0316,Y -123.4951,Z 164,A -116.4083,B 11.8425,C 0.2768,E1 11.7718,E2 207.0586} C_DIS
LIN {X -62.7034,Y -125.218,Z 164,A -114.8773,B 11.8425,C 0.2788,E1 11.7756,E2 205.528} C_DIS
LIN {X -59.1002,Y -126.9562,Z 164,A -113.2402,B 11.8424,C 0.2806,E1 11.7798,E2 203.8909} C_DIS
LIN {X -55.9033,Y -128.396,Z 164,A -111.7982,B 11.8424,C 0.282,E1 11.7835,E2 202.4479} C_DIS
LIN {X -52.6923,Y -129.7469,Z 164,A -110.3677,B 11.8424,C 0.2833,E1 11.7872,E2 201.0167} C_DIS
LIN {X -49.4606,Y -131.0129,Z 164,A -108.901,B 11.8424,C 0.2834,E1 11.791,E2 199.5439} C_DIS
LIN {X -46.2108,Y -132.1942,Z 164,A -107.5239,B 11.8423,C 0.2856,E1 11.7946,E2 198.1715} C_DIS
LIN {X -42.9447,Y -133.291,Z 164,A -106.1105,B 11.8423,C 0.2866,E1 11.7984,E2 196.7574} C_DIS
LIN {X -39.6673,Y -134.3028,Z 164,A -104.6987,B 11.8423,C 0.2874,E1 11.8021,E2 195.3444} C_DIS
LIN {X -36.3902,Y -135.2276,Z 164,A -103.3057,B 11.8423,C 0.2883,E1 11.8059,E2 193.9511} C_DIS
LIN {X -33.0898,Y -136.0728,Z 164,A -101.9098,B 11.8422,C 0.2891,E1 11.8097,E2 192.5547} C_DIS
LIN {X -29.7983,Y -136.8312,Z 164,A -100.5291,B 11.8422,C 0.2899,E1 11.8134,E2 191.1738} C_DIS
LIN {X -26.5137,Y -137.5054,Z 164,A -99.1633,B 11.8422,C 0.2906,E1 11.8172,E2 189.8084} C_DIS
LIN {X -23.4452,Y -138.0622,Z 164,A -98.0238,B 11.842,C 0.2947,E1 11.8203,E2 188.6864} C_DIS
LIN {X -20.5352,Y -138.5263,Z 164,A -96.6499,B 11.8421,C 0.2907,E1 11.8241,E2 187.2902} C_DIS
LIN {X -17.1213,Y -138.9887,Z 164,A -95.2414,B 11.8421,C 0.291,E1 11.828,E2 185.8814} C_DIS
LIN {X -13.7009,Y -139.3668,Z 164,A -93.7486,B 11.8421,C 0.289,E1 11.8322,E2 184.3769} C_DIS
LIN {X -9.8203,Y -139.694,Z 164,A -92.1149,B 11.8422,C 0.2881,E1 11.8368,E2 182.7373} C_DIS
LIN {X -5.1239,Y -139.945,Z 164,A -90.3249,B 11.8422,C 0.2917,E1 11.8417,E2 180.9641} C_DIS
LIN {X -1.6056,Y -140.031,Z 164,A -88.7583,B 11.8422,C 0.2881,E1 11.8461,E2 179.3803} C_DIS
LIN {X -1.6056,Y -140.031,Z 164,A -88.7583,B 11.8422,C 0.2881,E1 11.8461,E2 179.3803} C_DIS
Enddeposition()
LIN {X 0.9509,Y -131.0535,Z 165,A -88.5381,B 12.0255,C 0.227,E1 12.0295,E2 178.8578} C_DIS
Startdeposition()
$VEL.CP = VEL_PRINT
LIN {X -1.6137,Y -131.0491,Z 165,A -89.9514,B 12.0253,C 0.2345,E1 12.0255,E2 180.3067} C_DIS
LIN {X -5.6075,Y -130.9387,Z 165,A -91.705,B 12.0253,C 0.2347,E1 12.0206,E2 182.0619} C_DIS
LIN {X -8.8735,Y -130.7586,Z 165,A -93.1154,B 12.0253,C 0.2342,E1 12.0166,E2 183.4705} C_DIS
LIN {X -12.8505,Y -130.4265,Z 165,A -94.8473,B 12.0253,C 0.2336,E1 12.0118,E2 185.2015} C_DIS
LIN {X -16.0462,Y -130.0726,Z 165,A -96.2509,B 12.0253,C 0.2333,E1 12.0079,E2 186.6055} C_DIS
LIN {X -19.2305,Y -129.6409,Z 165,A -97.7996,B 12.0253,C 0.2364,E1 12.0036,E2 188.1718} C_DIS
LIN {X -22.4144,Y -129.1284,Z 165,A -99.1266,B 12.0253,C 0.2339,E1 12,E2 189.4893} C_DIS
LIN {X -25.5718,Y -128.5398,Z 165,A -100.4953,B 12.0253,C 0.2324,E1 11.9962,E2 190.8541} C_DIS
LIN {X -29.3402,Y -127.7311,Z 165,A -102.2372,B 12.0253,C 0.2329,E1 11.9915,E2 192.6032} C_DIS
LIN {X -33.4124,Y -126.7272,Z 165,A -104.0435,B 12.0253,C 0.2312,E1 11.9866,E2 194.4066} C_DIS
LIN {X -37.3127,Y -125.6346,Z 165,A -105.7877,B 12.0254,C 0.2293,E1 11.9819,E2 196.1479} C_DIS
LIN {X -40.3432,Y -124.6944,Z 165,A -107.183,B 12.0254,C 0.2285,E1 11.9782,E2 197.5444} C_DIS
LIN {X -43.3855,Y -123.6687,Z 165,A -108.6341,B 12.0254,C 0.2285,E1 11.9743,E2 199.0013} C_DIS
LIN {X -47.1684,Y -122.2754,Z 165,A -110.3599,B 12.0254,C 0.2259,E1 11.9698,E2 200.7228} C_DIS
LIN {X -50.1517,Y -121.0824,Z 165,A -111.7722,B 12.0255,C 0.2247,E1 11.9662,E2 202.1361} C_DIS
LIN {X -53.1135,Y -119.8129,Z 165,A -113.2492,B 12.0255,C 0.2249,E1 11.9624,E2 203.6212} C_DIS
LIN {X -56.8242,Y -118.0979,Z 165,A -115.1115,B 12.0255,C 0.2246,E1 11.9577,E2 205.4923} C_DIS
LIN {X -60.3649,Y -116.3291,Z 165,A -116.6975,B 12.0256,C 0.2191,E1 11.9538,E2 207.0612} C_DIS
LIN {X -63.8844,Y -114.4353,Z 165,A -118.4839,B 12.0256,C 0.2177,E1 11.9494,E2 208.8521} C_DIS
LIN {X -67.3734,Y -112.4163,Z 165,A -120.2583,B 12.0256,C 0.2156,E1 11.9451,E2 210.6277} C_DIS
LIN {X -70.1204,Y -110.7234,Z 165,A -121.8313,B 12.0256,C 0.2173,E1 11.9413,E2 212.2196} C_DIS
LIN {X -73.5137,Y -108.5,Z 165,A -123.6085,B 12.0256,C 0.2146,E1 11.9372,E2 213.9969} C_DIS
LIN {X -77.4325,Y -105.7391,Z 165,A -125.7196,B 12.0257,C 0.2116,E1 11.9324,E2 216.1092} C_DIS
LIN {X -80.6347,Y -103.3185,Z 165,A -127.4917,B 12.0257,C 0.209,E1 11.9285,E2 217.883} C_DIS
LIN {X -84.167,Y -100.4611,Z 165,A -129.4016,B 12.0259,C 0.2037,E1 11.9244,E2 219.7831} C_DIS
LIN {X -87.1176,Y -97.9142,Z 165,A -131.1515,B 12.0259,C 0.2016,E1 11.9207,E2 221.5379} C_DIS
LIN {X -90.0772,Y -95.1979,Z 165,A -132.8993,B 12.0259,C 0.1981,E1 11.9171,E2 223.284} C_DIS
LIN {X -92.9515,Y -92.3933,Z 165,A -134.6703,B 12.026,C 0.1949,E1 11.9136,E2 225.0561} C_DIS
LIN {X -95.7786,Y -89.4594,Z 165,A -136.4951,B 12.026,C 0.1922,E1 11.9101,E2 226.8851} C_DIS
LIN {X -98.5039,Y -86.4501,Z 165,A -138.3387,B 12.026,C 0.19,E1 11.9067,E2 228.7359} C_DIS
LIN {X -100.4771,Y -84.1479,Z 165,A -139.617,B 12.0262,C 0.186,E1 11.9044,E2 230.008} C_DIS
LIN {X -103.0827,Y -80.935,Z 165,A -141.4152,B 12.0262,C 0.1818,E1 11.9012,E2 231.804} C_DIS
LIN {X -105.7363,Y -77.4363,Z 165,A -143.3684,B 12.0262,C 0.1781,E1 11.898,E2 233.7601} C_DIS
LIN {X -108.0763,Y -74.1352,Z 165,A -145.2277,B 12.0263,C 0.1759,E1 11.895,E2 235.6289} C_DIS
LIN {X -110.2796,Y -70.8163,Z 165,A -146.8336,B 12.0264,C 0.1688,E1 11.8925,E2 237.2177} C_DIS
LIN {X -111.9877,Y -68.0835,Z 165,A -148.2599,B 12.0264,C 0.1657,E1 11.8905,E2 238.6451} C_DIS
LIN {X -113.6342,Y -65.2989,Z 165,A -149.6968,B 12.0264,C 0.1626,E1 11.8884,E2 240.0838} C_DIS
LIN {X -115.5866,Y -61.7764,Z 165,A -151.4921,B 12.0265,C 0.1589,E1 11.886,E2 241.8819} C_DIS
LIN {X -117.3609,Y -58.3314,Z 165,A -153.218,B 12.0265,C 0.1552,E1 11.8838,E2 243.6101} C_DIS
LIN {X -118.8283,Y -55.2804,Z 165,A -154.6726,B 12.0266,C 0.1508,E1 11.8821,E2 245.0606} C_DIS
LIN {X -120.3214,Y -51.9496,Z 165,A -156.3461,B 12.0266,C 0.1482,E1 11.8802,E2 246.7419} C_DIS
LIN {X -121.6912,Y -48.6559,Z 165,A -157.8718,B 12.0267,C 0.1433,E1 11.8786,E2 248.2624} C_DIS
LIN {X -122.8474,Y -45.6578,Z 165,A -159.2925,B 12.0267,C 0.1398,E1 11.8772,E2 249.6838} C_DIS
LIN {X -123.9299,Y -42.632,Z 165,A -160.7134,B 12.0268,C 0.1363,E1 11.8759,E2 251.1053} C_DIS
LIN {X -124.9377,Y -39.5815,Z 165,A -162.1368,B 12.0268,C 0.1328,E1 11.8747,E2 252.5297} C_DIS
LIN {X -125.8763,Y -36.487,Z 165,A -163.564,B 12.0268,C 0.1291,E1 11.8735,E2 253.9571} C_DIS
LIN {X -126.9306,Y -32.6316,Z 165,A -165.4939,B 12.0269,C 0.1281,E1 11.8721,E2 255.9067} C_DIS
LIN {X -127.8737,Y -28.7158,Z 165,A -167.114,B 12.0269,C 0.1201,E1 11.8711,E2 257.5088} C_DIS
LIN {X -128.544,Y -25.5509,Z 165,A -168.5407,B 12.027,C 0.1163,E1 11.8703,E2 258.9356} C_DIS
LIN {X -129.1601,Y -22.2307,Z 165,A -169.9923,B 12.027,C 0.1115,E1 11.8696,E2 260.3829} C_DIS
LIN {X -129.6383,Y -19.2484,Z 165,A -171.3926,B 12.027,C 0.1094,E1 11.869,E2 261.7913} C_DIS
LIN {X -130.125,Y -15.607,Z 165,A -173.0652,B 12.0271,C 0.1061,E1 11.8684,E2 263.4698} C_DIS
LIN {X -130.5024,Y -12.0598,Z 165,A -174.5761,B 12.0271,C 0.1005,E1 11.868,E2 264.9735} C_DIS
LIN {X -130.7597,Y -8.8584,Z 165,A -176.0113,B 12.0271,C 0.097,E1 11.8677,E2 266.4109} C_DIS
LIN {X -130.9385,Y -5.6115,Z 165,A -177.6121,B 12.0271,C 0.0966,E1 11.8675,E2 268.031} C_DIS
LIN {X -131.0504,Y -1.533,Z 165,A -179.1643,B 12.0273,C 0.0865,E1 11.8674,E2 269.5545} C_DIS
LIN {X -131.0354,Y 2.4316,Z 165,A 178.9984,B 12.0273,C 0.0835,E1 11.8674,E2 271.4019} C_DIS
LIN {X -130.9387,Y 5.6066,Z 165,A 177.597,B 12.0273,C 0.0797,E1 11.8676,E2 272.8033} C_DIS
LIN {X -130.7603,Y 8.8509,Z 165,A 176.1356,B 12.0273,C 0.0764,E1 11.8678,E2 274.268} C_DIS
LIN {X -130.5015,Y 12.0693,Z 165,A 174.6801,B 12.0273,C 0.0731,E1 11.8682,E2 275.7269} C_DIS
LIN {X -130.0673,Y 16.0906,Z 165,A 172.935,B 12.0273,C 0.0675,E1 11.8687,E2 277.4673} C_DIS
LIN {X -129.6365,Y 19.2614,Z 165,A 171.5064,B 12.0274,C 0.064,E1 11.8693,E2 278.8978} C_DIS
LIN {X -129.1273,Y 22.4202,Z 165,A 170.0799,B 12.0274,C 0.0605,E1 11.8699,E2 280.3259} C_DIS
LIN {X -128.5403,Y 25.5689,Z 165,A 168.6644,B 12.0274,C 0.0567,E1 11.8707,E2 281.7416} C_DIS
LIN {X -127.871,Y 28.7275,Z 165,A 167.2363,B 12.0274,C 0.0529,E1 11.8715,E2 283.1699} C_DIS
LIN {X -126.9259,Y 32.6503,Z 165,A 165.4567,B 12.0274,C 0.0482,E1 11.8727,E2 284.9493} C_DIS
LIN {X -126.0978,Y 35.7151,Z 165,A 164.0374,B 12.0274,C 0.0449,E1 11.8738,E2 286.3706} C_DIS
LIN {X -124.9384,Y 39.5794,Z 165,A 162.2628,B 12.0275,C 0.0401,E1 11.8752,E2 288.1444} C_DIS
LIN {X -123.9305,Y 42.6304,Z 165,A 160.8412,B 12.0275,C 0.0365,E1 11.8765,E2 289.5663} C_DIS
LIN {X -122.8483,Y 45.6555,Z 165,A 159.3944,B 12.0275,C 0.0334,E1 11.8779,E2 291.0163} C_DIS
LIN {X -121.6526,Y 48.7517,Z 165,A 157.8434,B 12.0275,C 0.0315,E1 11.8795,E2 292.5772} C_DIS
LIN {X -120.1244,Y 52.4052,Z 165,A 156.0477,B 12.0275,C 0.0281,E1 11.8815,E2 294.3782} C_DIS
LIN {X -118.4282,Y 56.133,Z 165,A 154.4246,B 12.0275,C 0.0197,E1 11.8833,E2 295.9799} C_DIS
LIN {X -117.0628,Y 58.929,Z 165,A 152.8959,B 12.0275,C 0.0197,E1 11.8853,E2 297.5265} C_DIS
LIN {X -115.2133,Y 62.4702,Z 165,A 151.1457,B 12.0275,C 0.0151,E1 11.8876,E2 299.2751} C_DIS
LIN {X -113.004,Y 66.3822,Z 165,A 149.1484,B 12.0275,C 0.0107,E1 11.8903,E2 301.2739} C_DIS
LIN {X -110.6903,Y 70.1729,Z 165,A 147.138,B 12.0275,C 0.0072,E1 11.8933,E2 303.29} C_DIS
LIN {X -108.0664,Y 74.1496,Z 165,A 145.1896,B 12.0275,C -0.0009,E1 11.8963,E2 305.2205} C_DIS
LIN {X -106.2158,Y 76.7772,Z 165,A 143.7727,B 12.0275,C -0.004,E1 11.8986,E2 306.6372} C_DIS
LIN {X -103.8133,Y 79.9965,Z 165,A 141.8997,B 12.0275,C -0.0057,E1 11.9018,E2 308.5216} C_DIS
LIN {X -101.3038,Y 83.1512,Z 165,A 140.1352,B 12.0275,C -0.0098,E1 11.9049,E2 310.2844} C_DIS
LIN {X -98.709,Y 86.215,Z 165,A 138.3762,B 12.0275,C -0.0138,E1 11.9081,E2 312.0418} C_DIS
LIN {X -96.0211,Y 89.1991,Z 165,A 136.5901,B 12.0275,C -0.017,E1 11.9114,E2 313.8295} C_DIS
LIN {X -93.2315,Y 92.1115,Z 165,A 134.7944,B 12.0275,C -0.0201,E1 11.9149,E2 315.627} C_DIS
LIN {X -90.3661,Y 94.9238,Z 165,A 133.0416,B 12.0275,C -0.0239,E1 11.9185,E2 317.3776} C_DIS
LIN {X -87.4154,Y 97.6476,Z 165,A 131.2798,B 12.0275,C -0.0273,E1 11.9221,E2 319.1383} C_DIS
LIN {X -84.3827,Y 100.2801,Z 165,A 129.4931,B 12.0275,C -0.0301,E1 11.9259,E2 320.9267} C_DIS
LIN {X -81.2592,Y 102.828,Z 165,A 127.707,B 12.0275,C -0.0329,E1 11.9298,E2 322.7138} C_DIS
LIN {X -78.071,Y 105.2686,Z 165,A 125.8698,B 12.0275,C -0.0343,E1 11.9339,E2 324.5585} C_DIS
LIN {X -74.8244,Y 107.6003,Z 165,A 124.2685,B 12.0275,C -0.0406,E1 11.9375,E2 326.1413} C_DIS
LIN {X -72.1636,Y 109.4026,Z 165,A 122.8522,B 12.0275,C -0.0428,E1 11.9408,E2 327.5575} C_DIS
LIN {X -69.3088,Y 111.2331,Z 165,A 121.2247,B 12.0275,C -0.0419,E1 11.9447,E2 329.2002} C_DIS
LIN {X -65.2672,Y 113.6523,Z 165,A 119.2848,B 12.0275,C -0.0478,E1 11.9493,E2 331.1245} C_DIS
LIN {X -61.7655,Y 115.5925,Z 165,A 117.5027,B 12.0275,C -0.0497,E1 11.9537,E2 332.9086} C_DIS
LIN {X -58.9224,Y 117.0662,Z 165,A 116.1107,B 12.0275,C -0.0518,E1 11.9571,E2 334.2984} C_DIS
LIN {X -56.0415,Y 118.4719,Z 165,A 114.5806,B 12.0275,C -0.0508,E1 11.961,E2 335.842} C_DIS
LIN {X -52.381,Y 120.1349,Z 165,A 112.9433,B 12.0275,C -0.0557,E1 11.9652,E2 337.464} C_DIS
LIN {X -49.4227,Y 121.3821,Z 165,A 111.532,B 12.0275,C -0.0572,E1 11.9688,E2 338.875} C_DIS
LIN {X -46.3973,Y 122.5704,Z 165,A 110.1111,B 12.0275,C -0.0588,E1 11.9725,E2 340.2947} C_DIS
LIN {X -42.8815,Y 123.8434,Z 165,A 108.4149,B 12.0275,C -0.0591,E1 11.977,E2 341.9966} C_DIS
LIN {X -39.5662,Y 124.9426,Z 165,A 106.927,B 12.0275,C -0.0615,E1 11.9809,E2 343.479} C_DIS
LIN {X -36.4956,Y 125.8738,Z 165,A 105.5195,B 12.0275,C -0.0627,E1 11.9847,E2 344.8859} C_DIS
LIN {X -32.6452,Y 126.9272,Z 165,A 103.6061,B 12.0275,C -0.0602,E1 11.9899,E2 346.8173} C_DIS
LIN {X -28.7277,Y 127.871,Z 165,A 102.0047,B 12.0274,C -0.0652,E1 11.9942,E2 348.3992} C_DIS
LIN {X -25.27,Y 128.5999,Z 165,A 100.3062,B 12.0274,C -0.0626,E1 11.9989,E2 350.1143} C_DIS
LIN {X -21.58,Y 129.2686,Z 165,A 98.8071,B 12.0274,C -0.0668,E1 12.003,E2 351.5962} C_DIS
LIN {X -18.4432,Y 129.7534,Z 165,A 97.4185,B 12.0274,C -0.0675,E1 12.0068,E2 352.9841} C_DIS
LIN {X -15.219,Y 130.1713,Z 165,A 96.0042,B 12.0274,C -0.0683,E1 12.0107,E2 354.3967} C_DIS
LIN {X -12.06,Y 130.5024,Z 165,A 94.6122,B 12.0274,C -0.0687,E1 12.0146,E2 355.7883} C_DIS
LIN {X -8.8368,Y 130.7613,Z 165,A 93.178,B 12.0274,C -0.0686,E1 12.0186,E2 357.2241} C_DIS
LIN {X -4.9251,Y 130.9653,Z 165,A 91.4677,B 12.0274,C -0.069,E1 12.0233,E2 358.9333} C_DIS
LIN {X -1.6043,Y 131.0492,Z 165,A 90.0422,B 12.0274,C -0.0698,E1 12.0273,E2 360.355} C_DIS
LIN {X 1.61,Y 131.0492,Z 165,A 88.4379,B 12.0274,C -0.065,E1 12.0319,E2 361.9815} C_DIS
LIN {X 5.6219,Y 130.9381,Z 165,A 86.8745,B 12.0274,C -0.0696,E1 12.0362,E2 363.5222} C_DIS
LIN {X 8.8662,Y 130.7592,Z 165,A 85.4332,B 12.0274,C -0.0689,E1 12.0402,E2 364.9654} C_DIS
LIN {X 12.0692,Y 130.5015,Z 165,A 83.8791,B 12.0274,C -0.065,E1 12.0445,E2 366.5361} C_DIS
LIN {X 16.0435,Y 130.0729,Z 165,A 82.3011,B 12.0274,C -0.0686,E1 12.0489,E2 368.0939} C_DIS
LIN {X 19.2372,Y 129.6399,Z 165,A 80.8893,B 12.0274,C -0.0681,E1 12.0528,E2 369.5058} C_DIS
LIN {X 22.4101,Y 129.1291,Z 165,A 79.4697,B 12.0274,C -0.0671,E1 12.0567,E2 370.9266} C_DIS
LIN {X 26.2384,Y 128.4041,Z 165,A 77.7572,B 12.0274,C -0.066,E1 12.0614,E2 372.6397} C_DIS
LIN {X 29.4989,Y 127.6948,Z 165,A 76.3244,B 12.0274,C -0.0658,E1 12.0653,E2 374.0692} C_DIS
LIN {X 33.4,Y 126.7305,Z 165,A 74.5658,B 12.0274,C -0.0646,E1 12.07,E2 375.8276} C_DIS
LIN {X 36.5131,Y 125.8687,Z 165,A 73.1642,B 12.0274,C -0.0638,E1 12.0738,E2 377.2278} C_DIS
LIN {X 39.587,Y 124.9359,Z 165,A 71.7657,B 12.0274,C -0.0628,E1 12.0775,E2 378.6255} C_DIS
LIN {X 42.6376,Y 123.928,Z 165,A 70.3667,B 12.0274,C -0.0617,E1 12.0812,E2 380.0236} C_DIS
LIN {X 45.6628,Y 122.8455,Z 165,A 68.9687,B 12.0274,C -0.0605,E1 12.0849,E2 381.4208} C_DIS
LIN {X 48.6696,Y 121.6856,Z 165,A 67.5665,B 12.0274,C -0.0593,E1 12.0885,E2 382.8222} C_DIS
LIN {X 52.0359,Y 120.2841,Z 165,A 66.0928,B 12.0274,C -0.0606,E1 12.0923,E2 384.2818} C_DIS
LIN {X 54.8733,Y 119.0165,Z 165,A 64.5383,B 12.0274,C -0.054,E1 12.0963,E2 385.8591} C_DIS
LIN {X 58.1979,Y 117.4268,Z 165,A 63.0211,B 12.0274,C -0.0544,E1 12.1001,E2 387.3655} C_DIS
LIN {X 61.1536,Y 115.915,Z 165,A 61.6773,B 12.0274,C -0.0553,E1 12.1034,E2 388.6969} C_DIS
LIN {X 63.8772,Y 114.4393,Z 165,A 60.1997,B 12.0274,C -0.0503,E1 12.107,E2 390.1891} C_DIS
LIN {X 67.3818,Y 112.4113,Z 165,A 58.4703,B 12.0274,C -0.0488,E1 12.1112,E2 391.9141} C_DIS
LIN {X 70.1674,Y 110.6937,Z 165,A 56.8947,B 12.0274,C -0.0429,E1 12.115,E2 393.5066} C_DIS
LIN {X 73.5011,Y 108.5085,Z 165,A 55.1701,B 12.0275,C -0.0406,E1 12.119,E2 395.2295} C_DIS
LIN {X 76.7777,Y 106.2154,Z 165,A 53.5903,B 12.0275,C -0.0421,E1 12.1225,E2 396.7902} C_DIS
LIN {X 79.9947,Y 103.8147,Z 165,A 51.7516,B 12.0275,C -0.0368,E1 12.1266,E2 398.6392} C_DIS
LIN {X 83.1367,Y 101.3156,Z 165,A 50.0244,B 12.0275,C -0.0344,E1 12.1304,E2 400.3637} C_DIS
LIN {X 86.2188,Y 98.7057,Z 165,A 48.2875,B 12.0275,C -0.0319,E1 12.1341,E2 402.0978} C_DIS
LIN {X 89.203,Y 96.0175,Z 165,A 46.5331,B 12.0275,C -0.0285,E1 12.1377,E2 403.8527} C_DIS
LIN {X 92.1035,Y 93.2394,Z 165,A 44.7754,B 12.0275,C -0.0249,E1 12.1412,E2 405.6114} C_DIS
LIN {X 94.9174,Y 90.3729,Z 165,A 43.0551,B 12.0275,C -0.0222,E1 12.1445,E2 407.3283} C_DIS
LIN {X 97.6414,Y 87.4223,Z 165,A 41.3038,B 12.0275,C -0.0186,E1 12.1478,E2 409.0798} C_DIS
LIN {X 100.5551,Y 84.0549,Z 165,A 39.3874,B 12.0275,C -0.0151,E1 12.1513,E2 410.9937} C_DIS
LIN {X 103.0811,Y 80.937,Z 165,A 37.657,B 12.0275,C -0.0118,E1 12.1543,E2 412.7223} C_DIS
LIN {X 105.7322,Y 77.4419,Z 165,A 35.8209,B 12.0275,C -0.0095,E1 12.1574,E2 414.55} C_DIS
LIN {X 108.006,Y 74.2375,Z 165,A 34.0995,B 12.0275,C -0.0053,E1 12.1601,E2 416.2728} C_DIS
LIN {X 110.2837,Y 70.8099,Z 165,A 32.3352,B 12.0275,C -0.0019,E1 12.1628,E2 418.0343} C_DIS
LIN {X 112.4246,Y 67.3595,Z 165,A 30.4405,B 12.0275,C 0.0058,E1 12.1656,E2 419.9441} C_DIS
LIN {X 114.4419,Y 63.8726,Z 165,A 28.6871,B 12.0275,C 0.01,E1 12.168,E2 421.6979} C_DIS
LIN {X 116.3312,Y 60.3609,Z 165,A 27.1122,B 12.0275,C 0.01,E1 12.17,E2 423.2543} C_DIS
LIN {X 117.7806,Y 57.4805,Z 165,A 25.6878,B 12.0275,C 0.014,E1 12.1718,E2 424.6814} C_DIS
LIN {X 119.4942,Y 53.8261,Z 165,A 23.9945,B 12.0275,C 0.0167,E1 12.1738,E2 426.3677} C_DIS
LIN {X 120.7724,Y 50.8941,Z 165,A 22.6013,B 12.0275,C 0.0203,E1 12.1753,E2 427.7615} C_DIS
LIN {X 121.9823,Y 47.9223,Z 165,A 21.1037,B 12.0275,C 0.0267,E1 12.1769,E2 429.2714} C_DIS
LIN {X 123.3972,Y 44.1503,Z 165,A 19.4704,B 12.0275,C 0.0281,E1 12.1784,E2 430.8911} C_DIS
LIN {X 124.442,Y 41.1132,Z 165,A 18.0816,B 12.0275,C 0.0316,E1 12.1797,E2 432.2794} C_DIS
LIN {X 125.6141,Y 37.3828,Z 165,A 16.3024,B 12.0275,C 0.0383,E1 12.1811,E2 434.0683} C_DIS
LIN {X 126.7454,Y 33.3441,Z 165,A 14.4349,B 12.0275,C 0.0444,E1 12.1825,E2 435.9415} C_DIS
LIN {X 127.7006,Y 29.4738,Z 165,A 12.8676,B 12.0275,C 0.0445,E1 12.1835,E2 437.4898} C_DIS
LIN {X 128.3843,Y 26.3357,Z 165,A 11.4708,B 12.0275,C 0.0484,E1 12.1843,E2 438.887} C_DIS
LIN {X 128.9916,Y 23.1788,Z 165,A 10.0844,B 12.0275,C 0.0519,E1 12.185,E2 440.2726} C_DIS
LIN {X 129.5208,Y 20.0111,Z 165,A 8.7035,B 12.0275,C 0.0553,E1 12.1857,E2 441.6521} C_DIS
LIN {X 129.9699,Y 16.8504,Z 165,A 7.2977,B 12.0275,C 0.0597,E1 12.1862,E2 443.0605} C_DIS
LIN {X 130.4271,Y 12.8445,Z 165,A 5.5719,B 12.0275,C 0.0638,E1 12.1867,E2 444.7838} C_DIS
LIN {X 130.7025,Y 9.6426,Z 165,A 4.1907,B 12.0274,C 0.0673,E1 12.187,E2 446.1636} C_DIS
LIN {X 130.9173,Y 6.0844,Z 165,A 2.5597,B 12.0274,C 0.0739,E1 12.1873,E2 447.8049} C_DIS
LIN {X 131.0492,Y 1.6027,Z 165,A 0.7998,B 12.0274,C 0.0742,E1 12.1873,E2 449.5431} C_DIS
LIN {X 131.0354,Y -2.4318,Z 165,A -1.0144,B 12.0274,C 0.0808,E1 12.1873,E2 451.3652} C_DIS
LIN {X 130.9388,Y -5.6036,Z 165,A -2.3798,B 12.0273,C 0.0843,E1 12.1872,E2 452.7296} C_DIS
LIN {X 130.759,Y -8.8688,Z 165,A -3.8116,B 12.0273,C 0.0886,E1 12.1869,E2 454.1632} C_DIS
LIN {X 130.4267,Y -12.8483,Z 165,A -5.5224,B 12.0273,C 0.0928,E1 12.1865,E2 455.8719} C_DIS
LIN {X 130.073,Y -16.0435,Z 165,A -6.9071,B 12.0272,C 0.0963,E1 12.1861,E2 457.2556} C_DIS
LIN {X 129.6413,Y -19.2274,Z 165,A -8.2947,B 12.0272,C 0.1,E1 12.1855,E2 458.6429} C_DIS
LIN {X 129.131,Y -22.3996,Z 165,A -9.7071,B 12.0272,C 0.1044,E1 12.1849,E2 460.0578} C_DIS
LIN {X 128.525,Y -25.6444,Z 165,A -11.1124,B 12.0271,C 0.1075,E1 12.1841,E2 461.4602} C_DIS
LIN {X 127.8675,Y -28.7429,Z 165,A -12.5793,B 12.0271,C 0.1138,E1 12.1833,E2 462.9385} C_DIS
LIN {X 126.9231,Y -32.6615,Z 165,A -14.2238,B 12.0271,C 0.1157,E1 12.1822,E2 464.5711} C_DIS
LIN {X 126.0967,Y -35.719,Z 165,A -15.6142,B 12.027,C 0.1198,E1 12.1811,E2 465.9638} C_DIS
LIN {X 124.9396,Y -39.5757,Z 165,A -17.4309,B 12.027,C 0.1264,E1 12.1796,E2 467.7892} C_DIS
LIN {X 123.671,Y -43.3787,Z 165,A -19.0691,B 12.0269,C 0.1282,E1 12.1782,E2 469.4159} C_DIS
LIN {X 122.5207,Y -46.53,Z 165,A -20.6667,B 12.0269,C 0.136,E1 12.1766,E2 471.0309} C_DIS
LIN {X 121.081,Y -50.1552,Z 165,A -22.1972,B 12.0269,C 0.1359,E1 12.175,E2 472.5426} C_DIS
LIN {X 119.8155,Y -53.1077,Z 165,A -23.5999,B 12.0268,C 0.1397,E1 12.1734,E2 473.9467} C_DIS
LIN {X 118.4593,Y -56.068,Z 165,A -24.987,B 12.0268,C 0.1426,E1 12.1718,E2 475.3311} C_DIS
LIN {X 116.9233,Y -59.2031,Z 165,A -26.3979,B 12.0268,C 0.1435,E1 12.1701,E2 476.73} C_DIS
LIN {X 115.5843,Y -61.7808,Z 165,A -27.9001,B 12.0266,C 0.1533,E1 12.1681,E2 478.2615} C_DIS
LIN {X 113.6206,Y -65.3224,Z 165,A -29.6643,B 12.0266,C 0.1578,E1 12.1656,E2 480.0271} C_DIS
LIN {X 111.5762,Y -68.7556,Z 165,A -31.2411,B 12.0266,C 0.1577,E1 12.1634,E2 481.5857} C_DIS
LIN {X 109.8575,Y -71.4692,Z 165,A -32.6306,B 12.0266,C 0.1609,E1 12.1613,E2 482.975} C_DIS
LIN {X 108.063,Y -74.1545,Z 165,A -34.0896,B 12.0264,C 0.1657,E1 12.159,E2 484.4413} C_DIS
LIN {X 105.7287,Y -77.4466,Z 165,A -35.9141,B 12.0264,C 0.1717,E1 12.156,E2 486.275} C_DIS
LIN {X 103.0778,Y -80.9411,Z 165,A -37.7405,B 12.0264,C 0.1739,E1 12.1529,E2 488.0928} C_DIS
LIN {X 100.535,Y -84.0789,Z 165,A -39.4965,B 12.0263,C 0.1778,E1 12.1498,E2 489.8496} C_DIS
LIN {X 97.9149,Y -87.1169,Z 165,A -41.2459,B 12.0263,C 0.1817,E1 12.1466,E2 491.6004} C_DIS
LIN {X 95.2023,Y -90.0725,Z 165,A -42.9601,B 12.0262,C 0.1846,E1 12.1433,E2 493.3119} C_DIS
LIN {X 92.3789,Y -92.9658,Z 165,A -44.7092,B 12.0262,C 0.188,E1 12.1399,E2 495.0608} C_DIS
LIN {X 89.4915,Y -95.7488,Z 165,A -46.4607,B 12.0261,C 0.1916,E1 12.1363,E2 496.814} C_DIS
LIN {X 86.5197,Y -98.4428,Z 165,A -48.2062,B 12.0261,C 0.1951,E1 12.1327,E2 498.5604} C_DIS
LIN {X 83.4316,Y -101.0728,Z 165,A -49.9416,B 12.026,C 0.1976,E1 12.129,E2 500.2932} C_DIS
LIN {X 80.3134,Y -103.5677,Z 165,A -51.6736,B 12.026,C 0.2006,E1 12.1252,E2 502.0253} C_DIS
LIN {X 77.3564,Y -105.7949,Z 165,A -53.3565,B 12.0258,C 0.2053,E1 12.1214,E2 503.7177} C_DIS
LIN {X 73.5002,Y -108.5091,Z 165,A -55.3209,B 12.0258,C 0.2064,E1 12.1169,E2 505.6725} C_DIS
LIN {X 70.1107,Y -110.7295,Z 165,A -57.1627,B 12.0258,C 0.2113,E1 12.1125,E2 507.5244} C_DIS
LIN {X 66.6986,Y -112.8182,Z 165,A -58.7478,B 12.0258,C 0.2099,E1 12.1088,E2 509.0917} C_DIS
LIN {X 63.8823,Y -114.4364,Z 165,A -60.3198,B 12.0257,C 0.2161,E1 12.1049,E2 510.6832} C_DIS
LIN {X 60.3614,Y -116.3309,Z 165,A -61.9061,B 12.0257,C 0.2145,E1 12.101,E2 512.2518} C_DIS
LIN {X 57.491,Y -117.7755,Z 165,A -63.305,B 12.0257,C 0.2163,E1 12.0975,E2 513.6513} C_DIS
LIN {X 54.5605,Y -119.1611,Z 165,A -64.8636,B 12.0256,C 0.222,E1 12.0936,E2 515.228} C_DIS
LIN {X 50.8993,Y -120.7702,Z 165,A -66.4397,B 12.0256,C 0.2197,E1 12.0896,E2 516.785} C_DIS
LIN {X 47.3092,Y -122.2206,Z 165,A -68.1491,B 12.0256,C 0.2222,E1 12.0851,E2 518.4978} C_DIS
LIN {X 43.5521,Y -123.6109,Z 165,A -69.9329,B 12.0255,C 0.225,E1 12.0804,E2 520.287} C_DIS
LIN {X 40.3197,Y -124.7019,Z 165,A -71.387,B 12.0255,C 0.2256,E1 12.0766,E2 521.7378} C_DIS
LIN {X 36.4556,Y -125.8855,Z 165,A -73.2629,B 12.0255,C 0.2302,E1 12.0715,E2 523.6281} C_DIS
LIN {X 31.8389,Y -127.1318,Z 165,A -75.1921,B 12.0255,C 0.2279,E1 12.0663,E2 525.5396} C_DIS
LIN {X 28.5154,Y -127.9195,Z 165,A -76.844,B 12.0253,C 0.2331,E1 12.0618,E2 527.2115} C_DIS
LIN {X 24.7557,Y -128.6983,Z 165,A -78.3601,B 12.0254,C 0.2302,E1 12.0577,E2 528.7093} C_DIS
LIN {X 21.5936,Y -129.2664,Z 165,A -79.7589,B 12.0254,C 0.2309,E1 12.0538,E2 530.1083} C_DIS
LIN {X 18.4353,Y -129.7545,Z 165,A -81.1496,B 12.0254,C 0.2316,E1 12.05,E2 531.4992} C_DIS
LIN {X 15.2138,Y -130.1719,Z 165,A -82.5575,B 12.0254,C 0.232,E1 12.0461,E2 532.9065} C_DIS
LIN {X 12.0573,Y -130.5027,Z 165,A -83.9436,B 12.0254,C 0.2325,E1 12.0422,E2 534.2933} C_DIS
LIN {X 8.854,Y -130.7601,Z 165,A -85.3596,B 12.0254,C 0.2333,E1 12.0383,E2 535.7113} C_DIS
LIN {X 5.5884,Y -130.9394,Z 165,A -86.9411,B 12.0253,C 0.2375,E1 12.0338,E2 537.3117} C_DIS
LIN {X 1.5985,Y -131.0493,Z 165,A -88.5076,B 12.0253,C 0.2334,E1 12.0295,E2 538.8578} C_DIS
LIN {X 1.5985,Y -131.0493,Z 165,A -88.5076,B 12.0253,C 0.2334,E1 12.0295,E2 538.8578} C_DIS
Enddeposition()
LIN {X 0.9568,Y -131.9698,Z 165,A -88.5082,B 12.0253,C 0.2337,E1 12.0295,E2 538.86} C_DIS
Startdeposition()
$VEL.CP = VEL_PRINT
LIN {X 3.7062,Y -131.9238,Z 165,A -86.9249,B 12.0254,C 0.2236,E1 12.034,E2 537.2289} C_DIS
LIN {X 7.4321,Y -131.7681,Z 165,A -85.2246,B 12.0254,C 0.2211,E1 12.0387,E2 535.5179} C_DIS
LIN {X 11.483,Y -131.4758,Z 165,A -83.5364,B 12.0254,C 0.2223,E1 12.0434,E2 533.8379} C_DIS
LIN {X 15.4708,Y -131.0659,Z 165,A -81.7757,B 12.0254,C 0.221,E1 12.0483,E2 532.0736} C_DIS
LIN {X 19.5204,Y -130.5258,Z 165,A -80.0657,B 12.0254,C 0.2217,E1 12.053,E2 530.3704} C_DIS
LIN {X 22.9925,Y -129.9576,Z 165,A -78.5492,B 12.0254,C 0.221,E1 12.0572,E2 528.8541} C_DIS
LIN {X 27.1767,Y -129.149,Z 165,A -76.227,B 12.0257,C 0.2073,E1 12.0637,E2 526.4729} C_DIS
LIN {X 31.084,Y -128.2628,Z 165,A -75.1276,B 12.0254,C 0.2227,E1 12.0665,E2 525.4505} C_DIS
LIN {X 38.685,Y -126.1784,Z 165,A -71.5219,B 12.0256,C 0.2147,E1 12.0763,E2 521.82} C_DIS
LIN {X 41.4042,Y -125.3128,Z 165,A -70.1489,B 12.0256,C 0.2099,E1 12.0799,E2 520.4297} C_DIS
LIN {X 45.6802,Y -123.8194,Z 165,A -68.2944,B 12.0256,C 0.2107,E1 12.0848,E2 518.5873} C_DIS
LIN {X 49.1817,Y -122.4691,Z 165,A -66.7102,B 12.0256,C 0.2099,E1 12.0889,E2 517.0072} C_DIS
LIN {X 52.1206,Y -121.2477,Z 165,A -65.3309,B 12.0257,C 0.2082,E1 12.0924,E2 515.627} C_DIS
LIN {X 55.2483,Y -119.8546,Z 165,A -63.915,B 12.0257,C 0.2081,E1 12.096,E2 514.2183} C_DIS
LIN {X 57.888,Y -118.6034,Z 165,A -62.685,B 12.0257,C 0.2073,E1 12.0991,E2 512.9919} C_DIS
LIN {X 60.8982,Y -117.0861,Z 165,A -61.1352,B 12.0257,C 0.2028,E1 12.103,E2 511.4302} C_DIS
LIN {X 64.5263,Y -115.1277,Z 165,A -59.3239,B 12.0258,C 0.1995,E1 12.1074,E2 509.6146} C_DIS
LIN {X 68.131,Y -113.0319,Z 165,A -57.5011,B 12.0258,C 0.1962,E1 12.1118,E2 507.7886} C_DIS
LIN {X 71.0819,Y -111.1997,Z 165,A -55.9311,B 12.026,C 0.192,E1 12.1155,E2 506.2095} C_DIS
LIN {X 75.0224,Y -108.5809,Z 165,A -54.0074,B 12.026,C 0.192,E1 12.12,E2 504.2998} C_DIS
LIN {X 78.1116,Y -106.3794,Z 165,A -52.3444,B 12.026,C 0.1884,E1 12.1237,E2 502.633} C_DIS
LIN {X 81.5654,Y -103.755,Z 165,A -50.4424,B 12.026,C 0.1843,E1 12.1279,E2 500.7268} C_DIS
LIN {X 85.1554,Y -100.8302,Z 165,A -48.4806,B 12.0261,C 0.1817,E1 12.1321,E2 498.7688} C_DIS
LIN {X 88.2525,Y -98.1303,Z 165,A -46.74,B 12.0261,C 0.1792,E1 12.1358,E2 497.0315} C_DIS
LIN {X 91.3381,Y -95.2649,Z 165,A -45.1536,B 12.0261,C 0.182,E1 12.1389,E2 495.4726} C_DIS
LIN {X 93.3806,Y -93.2639,Z 165,A -43.6335,B 12.0263,C 0.1716,E1 12.142,E2 493.9171} C_DIS
LIN {X 96.4777,Y -90.056,Z 165,A -41.7609,B 12.0263,C 0.169,E1 12.1456,E2 492.0501} C_DIS
LIN {X 99.29,Y -86.9456,Z 165,A -39.9285,B 12.0263,C 0.1645,E1 12.149,E2 490.2142} C_DIS
LIN {X 102.5173,Y -83.1162,Z 165,A -37.7511,B 12.0264,C 0.1593,E1 12.1529,E2 488.0339} C_DIS
LIN {X 105.3829,Y -79.451,Z 165,A -35.8625,B 12.0264,C 0.158,E1 12.1561,E2 486.159} C_DIS
LIN {X 107.618,Y -76.3971,Z 165,A -34.1192,B 12.0265,C 0.1512,E1 12.159,E2 484.4015} C_DIS
LIN {X 110.2078,Y -72.6102,Z 165,A -32.1884,B 12.0265,C 0.1479,E1 12.162,E2 482.4758} C_DIS
LIN {X 112.6943,Y -68.6887,Z 165,A -30.2295,B 12.0266,C 0.1443,E1 12.1648,E2 480.5215} C_DIS
LIN {X 114.0714,Y -66.3763,Z 165,A -28.667,B 12.0268,C 0.1301,E1 12.1671,E2 478.9095} C_DIS
LIN {X 116.1086,Y -62.7448,Z 165,A -27.2446,B 12.0268,C 0.1362,E1 12.1689,E2 477.5322} C_DIS
LIN {X 120.1622,Y -54.5813,Z 165,A -23.3168,B 12.0268,C 0.1263,E1 12.1737,E2 473.6034} C_DIS
LIN {X 121.6341,Y -51.2131,Z 165,A -21.901,B 12.0268,C 0.127,E1 12.1753,E2 472.2076} C_DIS
LIN {X 122.9292,Y -48.0204,Z 165,A -20.3378,B 12.0268,C 0.1209,E1 12.1769,E2 470.6344} C_DIS
LIN {X 124.2502,Y -44.4913,Z 165,A -18.7531,B 12.0269,C 0.1177,E1 12.1784,E2 469.054} C_DIS
LIN {X 125.7696,Y -39.9944,Z 165,A -16.6809,B 12.0269,C 0.1115,E1 12.1802,E2 466.978} C_DIS
LIN {X 127.0008,Y -35.8953,Z 165,A -14.8162,B 12.027,C 0.106,E1 12.1817,E2 465.1103} C_DIS
LIN {X 128.0719,Y -31.8672,Z 165,A -12.6484,B 12.0271,C 0.0906,E1 12.1832,E2 462.8967} C_DIS
LIN {X 128.9793,Y -27.9626,Z 165,A -11.4678,B 12.0271,C 0.1014,E1 12.1839,E2 461.7823} C_DIS
LIN {X 129.5851,Y -25.0062,Z 165,A -10.1257,B 12.0271,C 0.0967,E1 12.1846,E2 460.4348} C_DIS
LIN {X 130.1782,Y -21.7072,Z 165,A -8.6476,B 12.0271,C 0.0918,E1 12.1853,E2 458.9522} C_DIS
LIN {X 130.7309,Y -18.0928,Z 165,A -6.9943,B 12.0271,C 0.0852,E1 12.186,E2 457.2892} C_DIS
LIN {X 131.1819,Y -14.4576,Z 165,A -5.4772,B 12.0271,C 0.0826,E1 12.1865,E2 455.7792} C_DIS
LIN {X 131.522,Y -10.9364,Z 165,A -3.914,B 12.0272,C 0.0773,E1 12.1868,E2 454.2109} C_DIS
LIN {X 131.7941,Y -6.9296,Z 165,A -2.2372,B 12.0272,C 0.074,E1 12.1871,E2 452.5402} C_DIS
LIN {X 131.9423,Y -3.0418,Z 165,A -0.5039,B 12.0272,C 0.0678,E1 12.1873,E2 450.7998} C_DIS
LIN {X 131.9767,Y 0.4658,Z 165,A 0.9967,B 12.0273,C 0.0639,E1 12.1873,E2 449.3002} C_DIS
LIN {X 131.8866,Y 4.86,Z 165,A 2.8277,B 12.0273,C 0.0604,E1 12.1871,E2 447.4764} C_DIS
LIN {X 131.6633,Y 9.0908,Z 165,A 4.6876,B 12.0273,C 0.0545,E1 12.1868,E2 445.6122} C_DIS
LIN {X 131.3588,Y 12.7467,Z 165,A 6.1964,B 12.0273,C 0.0521,E1 12.1864,E2 444.1118} C_DIS
LIN {X 130.8938,Y 16.8663,Z 165,A 7.9911,B 12.0273,C 0.047,E1 12.1858,E2 442.3159} C_DIS
LIN {X 130.3505,Y 20.6528,Z 165,A 9.6715,B 12.0274,C 0.0416,E1 12.1851,E2 440.6315} C_DIS
LIN {X 129.741,Y 24.1908,Z 165,A 11.1099,B 12.0274,C 0.0405,E1 12.1844,E2 439.2061} C_DIS
LIN {X 129.1382,Y 27.2264,Z 165,A 12.5359,B 12.0274,C 0.0343,E1 12.1836,E2 437.7688} C_DIS
LIN {X 128.3013,Y 30.9243,Z 165,A 14.2536,B 12.0274,C 0.0276,E1 12.1825,E2 436.0408} C_DIS
LIN {X 126.2199,Y 38.5496,Z 165,A 17.5512,B 12.0274,C 0.0217,E1 12.18,E2 432.7564} C_DIS
LIN {X 124.9666,Y 42.444,Z 165,A 19.2743,B 12.0274,C 0.0182,E1 12.1785,E2 431.0382} C_DIS
LIN {X 123.7492,Y 45.8678,Z 165,A 20.8162,B 12.0274,C 0.0149,E1 12.177,E2 429.4991} C_DIS
LIN {X 122.466,Y 49.1894,Z 165,A 22.3003,B 12.0274,C 0.0124,E1 12.1755,E2 428.0212} C_DIS
LIN {X 121.1738,Y 52.2916,Z 165,A 23.7927,B 12.0274,C 0.0075,E1 12.1739,E2 426.5236} C_DIS
LIN {X 119.4452,Y 56.1338,Z 165,A 25.5534,B 12.0274,C 0.0046,E1 12.1718,E2 424.7697} C_DIS
LIN {X 117.5839,Y 59.9291,Z 165,A 27.4169,B 12.0274,C -0.001,E1 12.1695,E2 422.9013} C_DIS
LIN {X 115.6882,Y 63.5167,Z 165,A 29.2457,B 12.0274,C -0.0073,E1 12.1671,E2 421.0634} C_DIS
LIN {X 113.8904,Y 66.686,Z 165,A 30.9789,B 12.0274,C -0.0155,E1 12.1646,E2 419.3108} C_DIS
LIN {X 112.2109,Y 69.4752,Z 165,A 32.1926,B 12.0274,C -0.0135,E1 12.1628,E2 418.1202} C_DIS
LIN {X 109.8448,Y 73.1583,Z 165,A 33.9293,B 12.0274,C -0.0136,E1 12.1602,E2 416.4019} C_DIS
LIN {X 107.7721,Y 76.1787,Z 165,A 35.5654,B 12.0274,C -0.0187,E1 12.1576,E2 414.7594} C_DIS
LIN {X 105.5352,Y 79.2491,Z 165,A 37.2722,B 12.0274,C -0.0241,E1 12.1548,E2 413.0446} C_DIS
LIN {X 102.8297,Y 82.7289,Z 165,A 39.1489,B 12.0274,C -0.0274,E1 12.1515,E2 411.1713} C_DIS
LIN {X 100.0418,Y 86.0793,Z 165,A 41.0276,B 12.0274,C -0.0312,E1 12.1481,E2 409.2932} C_DIS
LIN {X 97.1547,Y 89.325,Z 165,A 42.8699,B 12.0274,C -0.0341,E1 12.1447,E2 407.4552} C_DIS
LIN {X 94.2678,Y 92.3666,Z 165,A 44.6928,B 12.0274,C -0.0379,E1 12.1411,E2 405.6312} C_DIS
LIN {X 91.0956,Y 95.4966,Z 165,A 46.6162,B 12.0274,C -0.0415,E1 12.1373,E2 403.7084} C_DIS
LIN {X 87.7728,Y 98.56,Z 165,A 48.5998,B 12.0274,C -0.0459,E1 12.1332,E2 401.7215} C_DIS
LIN {X 84.4654,Y 101.4088,Z 165,A 50.4669,B 12.0274,C -0.0486,E1 12.1292,E2 399.8571} C_DIS
LIN {X 81.0983,Y 104.1209,Z 165,A 52.3473,B 12.0274,C -0.0521,E1 12.1251,E2 397.9757} C_DIS
LIN {X 77.6159,Y 106.7418,Z 165,A 54.1512,B 12.0274,C -0.0529,E1 12.121,E2 396.1819} C_DIS
LIN {X 73.935,Y 109.3234,Z 165,A 56.4247,B 12.0274,C -0.0646,E1 12.1157,E2 393.8696} C_DIS
LIN {X 70.7953,Y 111.3831,Z 165,A 57.7777,B 12.0274,C -0.0598,E1 12.1126,E2 392.5493} C_DIS
LIN {X 66.9139,Y 113.7565,Z 165,A 59.728,B 12.0274,C -0.062,E1 12.1079,E2 390.6017} C_DIS
LIN {X 62.8234,Y 116.0663,Z 165,A 61.7939,B 12.0274,C -0.0655,E1 12.1029,E2 388.5323} C_DIS
LIN {X 59.1608,Y 117.975,Z 165,A 63.5726,B 12.0273,C -0.0674,E1 12.0985,E2 386.7552} C_DIS
LIN {X 56.1943,Y 119.4164,Z 165,A 65.092,B 12.0273,C -0.0714,E1 12.0946,E2 385.2254} C_DIS
LIN {X 52.1859,Y 121.2195,Z 165,A 66.7792,B 12.0273,C -0.0679,E1 12.0904,E2 383.5643} C_DIS
LIN {X 48.2375,Y 122.8448,Z 165,A 68.6311,B 12.0273,C -0.0698,E1 12.0856,E2 381.7127} C_DIS
LIN {X 44.724,Y 124.1663,Z 165,A 70.2214,B 12.0273,C -0.0703,E1 12.0814,E2 380.1272} C_DIS
LIN {X 41.0079,Y 125.4448,Z 165,A 72.0308,B 12.0273,C -0.0745,E1 12.0766,E2 378.3058} C_DIS
LIN {X 36.5731,Y 126.8078,Z 165,A 74.2439,B 12.0273,C -0.0811,E1 12.0706,E2 376.0693} C_DIS
LIN {X 33.2909,Y 127.7098,Z 165,A 75.4795,B 12.0273,C -0.076,E1 12.0673,E2 374.8628} C_DIS
LIN {X 30.5613,Y 128.3888,Z 165,A 76.9905,B 12.0272,C -0.0841,E1 12.0631,E2 373.3177} C_DIS
LIN {X 26.9594,Y 129.1943,Z 165,A 78.3127,B 12.0272,C -0.0779,E1 12.0596,E2 372.0291} C_DIS
LIN {X 23.0612,Y 129.9453,Z 165,A 79.9876,B 12.0272,C -0.0775,E1 12.055,E2 370.3604} C_DIS
LIN {X 18.8475,Y 130.6231,Z 165,A 81.8615,B 12.0272,C -0.0787,E1 12.0499,E2 368.4844} C_DIS
LIN {X 14.6048,Y 131.166,Z 165,A 83.7012,B 12.0272,C -0.0788,E1 12.0448,E2 366.6475} C_DIS
Enddeposition()
END
